LIN {X 0,Y 249.508,Z 932.66,A -85,B 0,C 180,E1 11833.837,E2 11833.837} C_VEL
LIN {X 0,Y 242.06,Z 946.637,A -85,B 0,C 180,E1 11830.431,E2 11830.431} C_VEL
LIN {X 0,Y 234.824,Z 959.705,A -85,B 0,C 180,E1 11826.415,E2 11826.415} C_VEL
LIN {X 0,Y 228.423,Z 971.273,A -85,B 0,C 180,E1 11821.878,E2 11821.878} C_VEL
LIN {X 0,Y 223.309,Z 980.961,A -85,B 0,C 180,E1 11817,E2 11817} C_VEL
LIN {X 0,Y 219.624,Z 988.763,A -85,B 0,C 180,E1 11811.922,E2 11811.922} C_VEL
LIN {X 0,Y 217.324,Z 994.963,A -85,B 0,C 180,E1 11806.575,E2 11806.575} C_VEL
LIN {X 0,Y 216.333,Z 999.398,A -85,B 0,C 180,E1 11801.195,E2 11801.195} C_VEL
LIN {X 0,Y 216.241,Z 1002.058,A -85,B 0,C 180,E1 11796.106,E2 11796.106} C_VEL
LIN {X 0,Y 216.392,Z 1003.045,A -85,B 0,C 180,E1 11791.59,E2 11791.59} C_VEL
LIN {X 0,Y 216.366,Z 1002.968,A -85,B 0,C 180,E1 11787.618,E2 11787.618} C_VEL
LIN {X 0,Y 216.189,Z 1001.566,A -85,B 0,C 180,E1 11782.828,E2 11782.828} C_VEL
LIN {X 0,Y 216.426,Z 998.664,A -85,B 0,C 180,E1 11777.732,E2 11777.732} C_VEL
LIN {X 0,Y 217.656,Z 993.876,A -85,B 0,C 180,E1 11772.352,E2 11772.352} C_VEL
LIN {X 0,Y 220.231,Z 987.265,A -85,B 0,C 180,E1 11767.019,E2 11767.019} C_VEL
LIN {X 0,Y 224.127,Z 979.16,A -85,B 0,C 180,E1 11762.042,E2 11762.042} C_VEL
LIN {X 0,Y 229.491,Z 969.097,A -85,B 0,C 180,E1 11757.231,E2 11757.231} C_VEL
LIN {X 0,Y 235.76,Z 957.78,A -85,B 0,C 180,E1 11752.972,E2 11752.972} C_VEL
LIN {X 0,Y 242.444,Z 945.727,A -85,B 0,C 180,E1 11749.339,E2 11749.339} C_VEL
LIN {X 0,Y 250.039,Z 931.432,A -85,B 0,C 180,E1 11745.911,E2 11745.911} C_VEL
LIN {X 0,Y 257.666,Z 916.125,A -85,B 0,C 180,E1 11742.993,E2 11742.993} C_VEL
LIN {X 0,Y 265.073,Z 899.972,A -85,B 0,C 180,E1 11740.532,E2 11740.532} C_VEL
LIN {X 0,Y 272.36,Z 882.29,A -85,B 0,C 180,E1 11738.394,E2 11738.394} C_VEL
LIN {X 0,Y 279.07,Z 863.665,A -85,B 0,C 180,E1 11736.627,E2 11736.627} C_VEL
LIN {X 0,Y 284.879,Z 844.815,A -85,B 0,C 180,E1 11735.245,E2 11735.245} C_VEL
LIN {X 0,Y 289.926,Z 824.777,A -85,B 0,C 180,E1 11734.141,E2 11734.141} C_VEL
LIN {X 0,Y 293.963,Z 803.375,A -85,B 0,C 180,E1 11733.295,E2 11733.295} C_VEL
LIN {X 0,Y 296.497,Z 782.175,A -85,B 0,C 180,E1 11732.711,E2 11732.711} C_VEL
LIN {X 0,Y 299.502,Z 753.951,A -85,B 0,C 180,E1 11732.36,E2 11732.36} C_VEL
LIN {X 0,Y 301.883,Z 735.107,A -85,B 0,C 180,E1 11732.253,E2 11732.253} C_VEL
LIN {X 0,Y 296.732,Z 710.347,A -85,B 0,C 180,E1 11729.497,E2 11729.497} C_VEL
LIN {X 0,Y 293.283,Z 686.164,A -85,B 0,C 180,E1 11727.059,E2 11727.059} C_VEL
LIN {X 0,Y 290.985,Z 658.881,A -85,B 0,C 180,E1 11724.649,E2 11724.649} C_VEL
LIN {X 0,Y 289.966,Z 631.512,A -85,B 0,C 180,E1 11722.557,E2 11722.557} C_VEL
LIN {X 0,Y 289.736,Z 625.924,A -85,B 0,C 180,E1 11722.095,E2 11722.095} C_VEL
LIN {X 0,Y 282.5,Z 605.873,A -85,B 0,C 180,E1 11716.553,E2 11716.553} C_VEL
LIN {X 0,Y 278.955,Z 593.643,A -85,B 0,C 180,E1 11712.629,E2 11712.629} C_VEL
LIN {X 0,Y 275.895,Z 578.468,A -85,B 0,C 180,E1 11706.817,E2 11706.817} C_VEL
LIN {X 0,Y 275.285,Z 568.562,A -85,B 0,C 180,E1 11702.289,E2 11702.289} C_VEL
LIN {X 0,Y 275.916,Z 561.635,A -85,B 0,C 180,E1 11698.65,E2 11698.65} C_VEL
LIN {X 0,Y 277.119,Z 556.907,A -85,B 0,C 180,E1 11695.758,E2 11695.758} C_VEL
LIN {X 0,Y 278.115,Z 554.651,A -85,B 0,C 180,E1 11694.015,E2 11694.015} C_VEL
LIN {X 0,Y 278.93,Z 555.456,A -85,B 0,C 180,E1 11692.378,E2 11692.378} C_VEL
LIN {X 0,Y 281.503,Z 559.555,A -85,B 0,C 180,E1 11688.527,E2 11688.527} C_VEL
LIN {X 0,Y 282.661,Z 561.038,A -85,B 0,C 180,E1 11687.227,E2 11687.227} C_VEL
LIN {X 0,Y 285.977,Z 565.926,A -85,B 0,C 180,E1 11684.07,E2 11684.07} C_VEL
LIN {X 0,Y 289.465,Z 571.159,A -85,B 0,C 180,E1 11681.366,E2 11681.366} C_VEL
LIN {X 0,Y 293.4,Z 577.167,A -85,B 0,C 180,E1 11678.772,E2 11678.772} C_VEL
LIN {X 0,Y 299.081,Z 586.337,A -85,B 0,C 180,E1 11675.562,E2 11675.562} C_VEL
LIN {X 0,Y 305.437,Z 597.593,A -85,B 0,C 180,E1 11672.458,E2 11672.458} C_VEL
LIN {X 0,Y 309.966,Z 606.51,A -85,B 0,C 180,E1 11670.461,E2 11670.461} C_VEL
LIN {X 0,Y 297.327,Z 772.309,A -85,B 0,C 180,E1 11666.864,E2 11666.864} C_VEL
LIN {X 0,Y 294.608,Z 792.529,A -85,B 0,C 180,E1 11666.172,E2 11666.172} C_VEL
LIN {X 0,Y 290.626,Z 813.159,A -85,B 0,C 180,E1 11665.173,E2 11665.173} C_VEL
LIN {X 0,Y 285.782,Z 832.475,A -85,B 0,C 180,E1 11663.918,E2 11663.918} C_VEL
LIN {X 0,Y 280.156,Z 850.837,A -85,B 0,C 180,E1 11662.389,E2 11662.389} C_VEL
LIN {X 0,Y 273.54,Z 869.084,A -85,B 0,C 180,E1 11660.465,E2 11660.465} C_VEL
LIN {X 0,Y 266.053,Z 886.914,A -85,B 0,C 180,E1 11658.081,E2 11658.081} C_VEL
LIN {X 0,Y 258.48,Z 902.921,A -85,B 0,C 180,E1 11655.376,E2 11655.376} C_VEL
LIN {X 0,Y 250.953,Z 917.393,A -85,B 0,C 180,E1 11652.324,E2 11652.324} C_VEL
LIN {X 0,Y 243.682,Z 930.447,A -85,B 0,C 180,E1 11648.885,E2 11648.885} C_VEL
LIN {X 0,Y 236.49,Z 942.746,A -85,B 0,C 180,E1 11644.802,E2 11644.802} C_VEL
LIN {X 0,Y 230.413,Z 952.929,A -85,B 0,C 180,E1 11640.51,E2 11640.51} C_VEL
LIN {X 0,Y 225.244,Z 961.693,A -85,B 0,C 180,E1 11635.785,E2 11635.785} C_VEL
LIN {X 0,Y 221.191,Z 968.962,A -85,B 0,C 180,E1 11630.644,E2 11630.644} C_VEL
LIN {X 0,Y 218.39,Z 974.6,A -85,B 0,C 180,E1 11625.126,E2 11625.126} C_VEL
LIN {X 0,Y 216.938,Z 978.219,A -85,B 0,C 180,E1 11619.817,E2 11619.817} C_VEL
LIN {X 0,Y 216.342,Z 980.279,A -85,B 0,C 180,E1 11614.505,E2 11614.505} C_VEL
LIN {X 0,Y 216.238,Z 980.863,A -85,B 0,C 180,E1 11609.469,E2 11609.469} C_VEL
LIN {X 0,Y 216.387,Z 980.118,A -85,B 0,C 180,E1 11604.696,E2 11604.696} C_VEL
LIN {X 0,Y 217.081,Z 977.836,A -85,B 0,C 180,E1 11599.382,E2 11599.382} C_VEL
LIN {X 0,Y 218.777,Z 973.736,A -85,B 0,C 180,E1 11593.811,E2 11593.811} C_VEL
LIN {X 0,Y 221.657,Z 968.101,A -85,B 0,C 180,E1 11588.568,E2 11588.568} C_VEL
LIN {X 0,Y 225.907,Z 960.633,A -85,B 0,C 180,E1 11583.446,E2 11583.446} C_VEL
LIN {X 0,Y 231.268,Z 951.656,A -85,B 0,C 180,E1 11578.746,E2 11578.746} C_VEL
LIN {X 0,Y 237.906,Z 940.55,A -85,B 0,C 180,E1 11574.253,E2 11574.253} C_VEL
LIN {X 0,Y 244.871,Z 928.525,A -85,B 0,C 180,E1 11570.431,E2 11570.431} C_VEL
LIN {X 0,Y 252.289,Z 915.077,A -85,B 0,C 180,E1 11567.025,E2 11567.025} C_VEL
LIN {X 0,Y 259.928,Z 900.139,A -85,B 0,C 180,E1 11563.999,E2 11563.999} C_VEL
LIN {X 0,Y 267.601,Z 883.56,A -85,B 0,C 180,E1 11561.32,E2 11561.32} C_VEL
LIN {X 0,Y 274.592,Z 866.606,A -85,B 0,C 180,E1 11559.14,E2 11559.14} C_VEL
LIN {X 0,Y 280.968,Z 848.815,A -85,B 0,C 180,E1 11557.31,E2 11557.31} C_VEL
LIN {X 0,Y 286.923,Z 828.967,A -85,B 0,C 180,E1 11555.711,E2 11555.711} C_VEL
LIN {X 0,Y 291.715,Z 808.912,A -85,B 0,C 180,E1 11554.478,E2 11554.478} C_VEL
LIN {X 0,Y 295.384,Z 788.518,A -85,B 0,C 180,E1 11553.556,E2 11553.556} C_VEL
LIN {X 0,Y 296.065,Z 783.376,A -85,B 0,C 180,E1 11553.352,E2 11553.352} C_VEL
LIN {X 0,Y 295.51,Z 784.886,A -85,B 0,C 180,E1 11553.294,E2 11553.294} C_VEL
LIN {X 0,Y 290.162,Z 799.608,A -85,B 0,C 180,E1 11552.949,E2 11552.949} C_VEL
LIN {X 0,Y 284.479,Z 812.877,A -85,B 0,C 180,E1 11552.694,E2 11552.694} C_VEL
LIN {X 0,Y 280.399,Z 820.06,A -85,B 0,C 180,E1 11552.37,E2 11552.37} C_VEL
LIN {X 0,Y 273.88,Z 829.294,A -85,B 0,C 180,E1 11551.593,E2 11551.593} C_VEL
LIN {X 0,Y 267.366,Z 836.64,A -85,B 0,C 180,E1 11550.571,E2 11550.571} C_VEL
LIN {X 0,Y 262.67,Z 841.252,A -85,B 0,C 180,E1 11549.66,E2 11549.66} C_VEL
LIN {X 0,Y 256.174,Z 848.136,A -85,B 0,C 180,E1 11548.573,E2 11548.573} C_VEL
LIN {X 0,Y 250.607,Z 852.992,A -85,B 0,C 180,E1 11547.311,E2 11547.311} C_VEL
LIN {X 0,Y 248.587,Z 854.447,A -85,B 0,C 180,E1 11546.775,E2 11546.775} C_VEL
LIN {X 0,Y 243.11,Z 859.517,A -85,B 0,C 180,E1 11545.585,E2 11545.585} C_VEL
LIN {X 0,Y 237.96,Z 863.392,A -85,B 0,C 180,E1 11544.053,E2 11544.053} C_VEL
LIN {X 0,Y 236.099,Z 864.688,A -85,B 0,C 180,E1 11543.459,E2 11543.459} C_VEL
LIN {X 0,Y 231.408,Z 868.479,A -85,B 0,C 180,E1 11542.081,E2 11542.081} C_VEL
LIN {X 0,Y 227.09,Z 871.222,A -85,B 0,C 180,E1 11540.308,E2 11540.308} C_VEL
LIN {X 0,Y 223.081,Z 874.46,A -85,B 0,C 180,E1 11538.827,E2 11538.827} C_VEL
LIN {X 0,Y 220.445,Z 875.936,A -85,B 0,C 180,E1 11537.419,E2 11537.419} C_VEL
LIN {X 0,Y 219.604,Z 876.415,A -85,B 0,C 180,E1 11536.942,E2 11536.942} C_VEL
LIN {X 0,Y 215.982,Z 879.302,A -85,B 0,C 180,E1 11535.3,E2 11535.3} C_VEL
LIN {X 0,Y 214.292,Z 880.186,A -85,B 0,C 180,E1 11534.042,E2 11534.042} C_VEL
LIN {X 0,Y 213.91,Z 880.409,A -85,B 0,C 180,E1 11533.516,E2 11533.516} C_VEL
LIN {X 0,Y 212.433,Z 891.843,A -85,B 0,C 180,E1 11529.756,E2 11529.756} C_VEL
LIN {X 0,Y 211.448,Z 902.388,A -85,B 0,C 180,E1 11525.427,E2 11525.427} C_VEL
LIN {X 0,Y 211.192,Z 910.701,A -85,B 0,C 180,E1 11521.086,E2 11521.086} C_VEL
LIN {X 0,Y 211.662,Z 917.257,A -85,B 0,C 180,E1 11516.751,E2 11516.751} C_VEL
LIN {X 0,Y 213.261,Z 922.908,A -85,B 0,C 180,E1 11511.604,E2 11511.604} C_VEL
LIN {X 0,Y 216.312,Z 926.54,A -85,B 0,C 180,E1 11506.365,E2 11506.365} C_VEL
LIN {X 0,Y 220.976,Z 928.025,A -85,B 0,C 180,E1 11501.261,E2 11501.261} C_VEL
LIN {X 0,Y 227.281,Z 927.461,A -85,B 0,C 180,E1 11496.402,E2 11496.402} C_VEL
LIN {X 0,Y 235.231,Z 924.927,A -85,B 0,C 180,E1 11491.849,E2 11491.849} C_VEL
LIN {X 0,Y 244.791,Z 920.464,A -85,B 0,C 180,E1 11487.651,E2 11487.651} C_VEL
LIN {X 0,Y 255.902,Z 914.126,A -85,B 0,C 180,E1 11483.844,E2 11483.844} C_VEL
LIN {X 0,Y 265.088,Z 908.328,A -85,B 0,C 180,E1 11481.246,E2 11481.246} C_VEL
LIN {X 0,Y 250.354,Z 921.045,A -85,B 0,C 180,E1 11477.635,E2 11477.635} C_VEL
LIN {X 0,Y 248.563,Z 923.055,A -85,B 0,C 180,E1 11477.065,E2 11477.065} C_VEL
LIN {X 0,Y 240.69,Z 937.7,A -85,B 0,C 180,E1 11473.929,E2 11473.929} C_VEL
LIN {X 0,Y 233.126,Z 950.904,A -85,B 0,C 180,E1 11470.365,E2 11470.365} C_VEL
LIN {X 0,Y 226.142,Z 962.79,A -85,B 0,C 180,E1 11466.334,E2 11466.334} C_VEL
LIN {X 0,Y 219.689,Z 973.857,A -85,B 0,C 180,E1 11461.562,E2 11461.562} C_VEL
LIN {X 0,Y 214.523,Z 983.296,A -85,B 0,C 180,E1 11456.283,E2 11456.283} C_VEL
LIN {X 0,Y 210.976,Z 990.727,A -85,B 0,C 180,E1 11450.822,E2 11450.822} C_VEL
LIN {X 0,Y 208.963,Z 996.327,A -85,B 0,C 180,E1 11445.26,E2 11445.26} C_VEL
LIN {X 0,Y 208.252,Z 999.989,A -85,B 0,C 180,E1 11439.955,E2 11439.955} C_VEL
LIN {X 0,Y 208.275,Z 1002.023,A -85,B 0,C 180,E1 11434.959,E2 11434.959} C_VEL
LIN {X 0,Y 208.42,Z 1002.729,A -85,B 0,C 180,E1 11430.551,E2 11430.551} C_VEL
LIN {X 0,Y 208.307,Z 1002.232,A -85,B 0,C 180,E1 11425.873,E2 11425.873} C_VEL
LIN {X 0,Y 208.203,Z 1000.547,A -85,B 0,C 180,E1 11421.162,E2 11421.162} C_VEL
LIN {X 0,Y 208.7,Z 997.166,A -85,B 0,C 180,E1 11415.859,E2 11415.859} C_VEL
LIN {X 0,Y 210.549,Z 991.635,A -85,B 0,C 180,E1 11410.008,E2 11410.008} C_VEL
LIN {X 0,Y 213.91,Z 984.361,A -85,B 0,C 180,E1 11404.437,E2 11404.437} C_VEL
LIN {X 0,Y 218.477,Z 975.891,A -85,B 0,C 180,E1 11399.472,E2 11399.472} C_VEL
LIN {X 0,Y 224.626,Z 965.286,A -85,B 0,C 180,E1 11394.645,E2 11394.645} C_VEL
LIN {X 0,Y 231.758,Z 953.089,A -85,B 0,C 180,E1 11390.321,E2 11390.321} C_VEL
LIN {X 0,Y 239.642,Z 939.321,A -85,B 0,C 180,E1 11386.496,E2 11386.496} C_VEL
LIN {X 0,Y 247.681,Z 924.434,A -85,B 0,C 180,E1 11383.228,E2 11383.228} C_VEL
LIN {X 0,Y 255.607,Z 908.668,A -85,B 0,C 180,E1 11380.492,E2 11380.492} C_VEL
LIN {X 0,Y 263.578,Z 891.117,A -85,B 0,C 180,E1 11378.084,E2 11378.084} C_VEL
LIN {X 0,Y 270.656,Z 873.481,A -85,B 0,C 180,E1 11376.18,E2 11376.18} C_VEL
LIN {X 0,Y 277.044,Z 855.14,A -85,B 0,C 180,E1 11374.63,E2 11374.63} C_VEL
LIN {X 0,Y 282.882,Z 835.046,A -85,B 0,C 180,E1 11373.34,E2 11373.34} C_VEL
LIN {X 0,Y 287.698,Z 813.932,A -85,B 0,C 180,E1 11372.359,E2 11372.359} C_VEL
LIN {X 0,Y 291.08,Z 792.615,A -85,B 0,C 180,E1 11371.65,E2 11371.65} C_VEL
LIN {X 0,Y 293.396,Z 770.364,A -85,B 0,C 180,E1 11371.208,E2 11371.208} C_VEL
LIN {X 0,Y 297.319,Z 737.114,A -85,B 0,C 180,E1 11370.937,E2 11370.937} C_VEL
LIN {X 0,Y 292.787,Z 713.367,A -85,B 0,C 180,E1 11368.269,E2 11368.269} C_VEL
LIN {X 0,Y 289.657,Z 689.519,A -85,B 0,C 180,E1 11365.822,E2 11365.822} C_VEL
LIN {X 0,Y 287.609,Z 661.966,A -85,B 0,C 180,E1 11363.348,E2 11363.348} C_VEL
LIN {X 0,Y 286.818,Z 634.141,A -85,B 0,C 180,E1 11361.189,E2 11361.189} C_VEL
LIN {X 0,Y 286.678,Z 630.805,A -85,B 0,C 180,E1 11360.892,E2 11360.892} C_VEL
LIN {X 0,Y 279.929,Z 610.615,A -85,B 0,C 180,E1 11355.167,E2 11355.167} C_VEL
LIN {X 0,Y 277.228,Z 600.398,A -85,B 0,C 180,E1 11351.81,E2 11351.81} C_VEL
LIN {X 0,Y 274.599,Z 585.5,A -85,B 0,C 180,E1 11346.061,E2 11346.061} C_VEL
LIN {X 0,Y 274.272,Z 575.732,A -85,B 0,C 180,E1 11341.566,E2 11341.566} C_VEL
LIN {X 0,Y 275.152,Z 568.696,A -85,B 0,C 180,E1 11337.836,E2 11337.836} C_VEL
LIN {X 0,Y 276.437,Z 564.313,A -85,B 0,C 180,E1 11335.124,E2 11335.124} C_VEL
LIN {X 0,Y 277.238,Z 562.671,A -85,B 0,C 180,E1 11333.788,E2 11333.788} C_VEL
LIN {X 0,Y 277.836,Z 563.406,A -85,B 0,C 180,E1 11332.556,E2 11332.556} C_VEL
LIN {X 0,Y 280.532,Z 567.621,A -85,B 0,C 180,E1 11328.487,E2 11328.487} C_VEL
LIN {X 0,Y 281.932,Z 569.872,A -85,B 0,C 180,E1 11326.881,E2 11326.881} C_VEL
LIN {X 0,Y 284.417,Z 573.484,A -85,B 0,C 180,E1 11324.503,E2 11324.503} C_VEL
LIN {X 0,Y 287.865,Z 578.85,A -85,B 0,C 180,E1 11321.731,E2 11321.731} C_VEL
LIN {X 0,Y 292.096,Z 585.427,A -85,B 0,C 180,E1 11318.883,E2 11318.883} C_VEL
LIN {X 0,Y 298.306,Z 596.028,A -85,B 0,C 180,E1 11315.336,E2 11315.336} C_VEL
LIN {X 0,Y 304.65,Z 607.99,A -85,B 0,C 180,E1 11312.222,E2 11312.222} C_VEL
LIN {X 0,Y 305.805,Z 610.542,A -85,B 0,C 180,E1 11311.685,E2 11311.685} C_VEL
LIN {X 0,Y 293.023,Z 772.739,A -85,B 0,C 180,E1 11308.171,E2 11308.171} C_VEL
LIN {X 0,Y 290.201,Z 793.084,A -85,B 0,C 180,E1 11307.476,E2 11307.476} C_VEL
LIN {X 0,Y 286.122,Z 813.58,A -85,B 0,C 180,E1 11306.486,E2 11306.486} C_VEL
LIN {X 0,Y 281.137,Z 832.867,A -85,B 0,C 180,E1 11305.238,E2 11305.238} C_VEL
LIN {X 0,Y 275.272,Z 851.399,A -85,B 0,C 180,E1 11303.696,E2 11303.696} C_VEL
LIN {X 0,Y 268.495,Z 869.487,A -85,B 0,C 180,E1 11301.788,E2 11301.788} C_VEL
LIN {X 0,Y 260.738,Z 887.322,A -85,B 0,C 180,E1 11299.399,E2 11299.399} C_VEL
LIN {X 0,Y 252.873,Z 903.332,A -85,B 0,C 180,E1 11296.678,E2 11296.678} C_VEL
LIN {X 0,Y 245.032,Z 917.806,A -85,B 0,C 180,E1 11293.597,E2 11293.597} C_VEL
LIN {X 0,Y 237.425,Z 930.862,A -85,B 0,C 180,E1 11290.113,E2 11290.113} C_VEL
LIN {X 0,Y 229.872,Z 943.163,A -85,B 0,C 180,E1 11285.957,E2 11285.957} C_VEL
LIN {X 0,Y 223.453,Z 953.346,A -85,B 0,C 180,E1 11281.567,E2 11281.567} C_VEL
LIN {X 0,Y 217.962,Z 962.111,A -85,B 0,C 180,E1 11276.714,E2 11276.714} C_VEL
LIN {X 0,Y 213.539,Z 969.52,A -85,B 0,C 180,E1 11271.285,E2 11271.285} C_VEL
LIN {X 0,Y 210.601,Z 975.016,A -85,B 0,C 180,E1 11265.699,E2 11265.699} C_VEL
LIN {X 0,Y 209.02,Z 978.633,A -85,B 0,C 180,E1 11260.193,E2 11260.193} C_VEL
LIN {X 0,Y 208.363,Z 980.691,A -85,B 0,C 180,E1 11254.678,E2 11254.678} C_VEL
LIN {X 0,Y 208.249,Z 981.275,A -85,B 0,C 180,E1 11249.448,E2 11249.448} C_VEL
LIN {X 0,Y 208.411,Z 980.53,A -85,B 0,C 180,E1 11244.492,E2 11244.492} C_VEL
LIN {X 0,Y 209.173,Z 978.25,A -85,B 0,C 180,E1 11238.976,E2 11238.976} C_VEL
LIN {X 0,Y 211.021,Z 974.151,A -85,B 0,C 180,E1 11233.199,E2 11233.199} C_VEL
LIN {X 0,Y 214.126,Z 968.516,A -85,B 0,C 180,E1 11227.774,E2 11227.774} C_VEL
LIN {X 0,Y 218.67,Z 961.049,A -85,B 0,C 180,E1 11222.494,E2 11222.494} C_VEL
LIN {X 0,Y 224.361,Z 952.07,A -85,B 0,C 180,E1 11217.67,E2 11217.67} C_VEL
LIN {X 0,Y 231.368,Z 940.962,A -85,B 0,C 180,E1 11213.079,E2 11213.079} C_VEL
LIN {X 0,Y 238.677,Z 928.935,A -85,B 0,C 180,E1 11209.191,E2 11209.191} C_VEL
LIN {X 0,Y 246.432,Z 915.484,A -85,B 0,C 180,E1 11205.742,E2 11205.742} C_VEL
LIN {X 0,Y 254.384,Z 900.542,A -85,B 0,C 180,E1 11202.691,E2 11202.691} C_VEL
LIN {X 0,Y 262.351,Z 883.958,A -85,B 0,C 180,E1 11199.999,E2 11199.999} C_VEL
LIN {X 0,Y 269.59,Z 866.998,A -85,B 0,C 180,E1 11197.815,E2 11197.815} C_VEL
LIN {X 0,Y 276.178,Z 849.2,A -85,B 0,C 180,E1 11195.986,E2 11195.986} C_VEL
LIN {X 0,Y 281.983,Z 830.511,A -85,B 0,C 180,E1 11194.475,E2 11194.475} C_VEL
LIN {X 0,Y 286.783,Z 811.098,A -85,B 0,C 180,E1 11193.247,E2 11193.247} C_VEL
LIN {X 0,Y 281.294,Z 818.614,A -85,B 0,C 180,E1 11192.462,E2 11192.462} C_VEL
LIN {X 0,Y 280.399,Z 820.06,A -85,B 0,C 180,E1 11192.37,E2 11192.37} C_VEL
LIN {X 0,Y 277.511,Z 825.438,A -85,B 0,C 180,E1 11192.229,E2 11192.229} C_VEL
LIN {X 0,Y 272.262,Z 836.502,A -85,B 0,C 180,E1 11192.306,E2 11192.306} C_VEL
LIN {X 0,Y 269.365,Z 840.573,A -85,B 0,C 180,E1 11192.061,E2 11192.061} C_VEL
LIN {X 0,Y 268.908,Z 841.051,A -85,B 0,C 180,E1 11191.993,E2 11191.993} C_VEL
LIN {X 0,Y 262.599,Z 846.992,A -85,B 0,C 180,E1 11190.932,E2 11190.932} C_VEL
LIN {X 0,Y 255.547,Z 854.023,A -85,B 0,C 180,E1 11189.796,E2 11189.796} C_VEL
LIN {X 0,Y 248.708,Z 859.476,A -85,B 0,C 180,E1 11188.32,E2 11188.32} C_VEL
LIN {X 0,Y 240.057,Z 866.645,A -85,B 0,C 180,E1 11186.425,E2 11186.425} C_VEL
LIN {X 0,Y 234.278,Z 870.564,A -85,B 0,C 180,E1 11184.724,E2 11184.724} C_VEL
LIN {X 0,Y 228.811,Z 874.703,A -85,B 0,C 180,E1 11183.159,E2 11183.159} C_VEL
LIN {X 0,Y 224.301,Z 877.414,A -85,B 0,C 180,E1 11181.441,E2 11181.441} C_VEL
LIN {X 0,Y 219.526,Z 880.861,A -85,B 0,C 180,E1 11179.697,E2 11179.697} C_VEL
LIN {X 0,Y 216.358,Z 882.596,A -85,B 0,C 180,E1 11178.037,E2 11178.037} C_VEL
LIN {X 0,Y 212.19,Z 885.615,A -85,B 0,C 180,E1 11176.142,E2 11176.142} C_VEL
LIN {X 0,Y 209.664,Z 886.901,A -85,B 0,C 180,E1 11174.359,E2 11174.359} C_VEL
LIN {X 0,Y 206.503,Z 889.328,A -85,B 0,C 180,E1 11172.585,E2 11172.585} C_VEL
LIN {X 0,Y 204.863,Z 890.186,A -85,B 0,C 180,E1 11170.973,E2 11170.973} C_VEL
LIN {X 0,Y 204.663,Z 890.482,A -85,B 0,C 180,E1 11170.55,E2 11170.55} C_VEL
LIN {X 0,Y 203.56,Z 901.222,A -85,B 0,C 180,E1 11166.204,E2 11166.204} C_VEL
LIN {X 0,Y 203.2,Z 910.642,A -85,B 0,C 180,E1 11161.41,E2 11161.41} C_VEL
LIN {X 0,Y 203.695,Z 917.877,A -85,B 0,C 180,E1 11156.624,E2 11156.624} C_VEL
LIN {X 0,Y 205.138,Z 923.3,A -85,B 0,C 180,E1 11151.875,E2 11151.875} C_VEL
LIN {X 0,Y 208.043,Z 927.408,A -85,B 0,C 180,E1 11146.663,E2 11146.663} C_VEL
LIN {X 0,Y 212.457,Z 929.549,A -85,B 0,C 180,E1 11141.621,E2 11141.621} C_VEL
LIN {X 0,Y 219.133,Z 929.77,A -85,B 0,C 180,E1 11136.327,E2 11136.327} C_VEL
LIN {X 0,Y 227.244,Z 928.012,A -85,B 0,C 180,E1 11131.629,E2 11131.629} C_VEL
LIN {X 0,Y 237.008,Z 924.384,A -85,B 0,C 180,E1 11127.318,E2 11127.318} C_VEL
LIN {X 0,Y 248.351,Z 918.964,A -85,B 0,C 180,E1 11123.428,E2 11123.428} C_VEL
LIN {X 0,Y 255.207,Z 915.31,A -85,B 0,C 180,E1 11121.428,E2 11121.428} C_VEL
LIN {X 0,Y 240.796,Z 926.761,A -85,B 0,C 180,E1 11117.658,E2 11117.658} C_VEL
LIN {X 0,Y 232.275,Z 941.595,A -85,B 0,C 180,E1 11114.217,E2 11114.217} C_VEL
LIN {X 0,Y 224.185,Z 954.904,A -85,B 0,C 180,E1 11110.295,E2 11110.295} C_VEL
LIN {X 0,Y 217.245,Z 966.132,A -85,B 0,C 180,E1 11106.096,E2 11106.096} C_VEL
LIN {X 0,Y 211.155,Z 976.06,A -85,B 0,C 180,E1 11101.392,E2 11101.392} C_VEL
LIN {X 0,Y 206.035,Z 984.955,A -85,B 0,C 180,E1 11095.899,E2 11095.899} C_VEL
LIN {X 0,Y 202.623,Z 991.877,A -85,B 0,C 180,E1 11090.209,E2 11090.209} C_VEL
LIN {X 0,Y 200.773,Z 996.99,A -85,B 0,C 180,E1 11084.42,E2 11084.42} C_VEL
LIN {X 0,Y 200.225,Z 1000.394,A -85,B 0,C 180,E1 11078.606,E2 11078.606} C_VEL
LIN {X 0,Y 200.334,Z 1001.972,A -85,B 0,C 180,E1 11073.722,E2 11073.722} C_VEL
LIN {X 0,Y 200.426,Z 1002.291,A -85,B 0,C 180,E1 11069.144,E2 11069.144} C_VEL
LIN {X 0,Y 200.262,Z 1001.527,A -85,B 0,C 180,E1 11064.558,E2 11064.558} C_VEL
LIN {X 0,Y 200.299,Z 999.213,A -85,B 0,C 180,E1 11059.067,E2 11059.067} C_VEL
LIN {X 0,Y 201.3,Z 995.149,A -85,B 0,C 180,E1 11053.258,E2 11053.258} C_VEL
LIN {X 0,Y 203.742,Z 989.322,A -85,B 0,C 180,E1 11047.495,E2 11047.495} C_VEL
LIN {X 0,Y 207.843,Z 981.57,A -85,B 0,C 180,E1 11041.874,E2 11041.874} C_VEL
LIN {X 0,Y 213.318,Z 972.31,A -85,B 0,C 180,E1 11036.744,E2 11036.744} C_VEL
LIN {X 0,Y 219.907,Z 961.632,A -85,B 0,C 180,E1 11032.136,E2 11032.136} C_VEL
LIN {X 0,Y 227.808,Z 948.812,A -85,B 0,C 180,E1 11027.817,E2 11027.817} C_VEL
LIN {X 0,Y 235.84,Z 935.273,A -85,B 0,C 180,E1 11024.237,E2 11024.237} C_VEL
LIN {X 0,Y 243.881,Z 920.882,A -85,B 0,C 180,E1 11021.211,E2 11021.211} C_VEL
LIN {X 0,Y 252.416,Z 904.235,A -85,B 0,C 180,E1 11018.455,E2 11018.455} C_VEL
LIN {X 0,Y 260.607,Z 886.289,A -85,B 0,C 180,E1 11016.138,E2 11016.138} C_VEL
LIN {X 0,Y 267.867,Z 868.033,A -85,B 0,C 180,E1 11014.307,E2 11014.307} C_VEL
LIN {X 0,Y 274.307,Z 849.121,A -85,B 0,C 180,E1 11012.843,E2 11012.843} C_VEL
LIN {X 0,Y 279.734,Z 829.887,A -85,B 0,C 180,E1 11011.715,E2 11011.715} C_VEL
LIN {X 0,Y 284.262,Z 809.32,A -85,B 0,C 180,E1 11010.833,E2 11010.833} C_VEL
LIN {X 0,Y 287.374,Z 788.684,A -85,B 0,C 180,E1 11010.188,E2 11010.188} C_VEL
LIN {X 0,Y 290.015,Z 763.795,A -85,B 0,C 180,E1 11009.782,E2 11009.782} C_VEL
LIN {X 0,Y 292.967,Z 739.242,A -85,B 0,C 180,E1 11009.604,E2 11009.604} C_VEL
LIN {X 0,Y 288.979,Z 716.38,A -85,B 0,C 180,E1 11007.008,E2 11007.008} C_VEL
LIN {X 0,Y 286.193,Z 693.135,A -85,B 0,C 180,E1 11004.58,E2 11004.58} C_VEL
LIN {X 0,Y 284.392,Z 665.207,A -85,B 0,C 180,E1 11002.029,E2 11002.029} C_VEL
LIN {X 0,Y 283.838,Z 636.802,A -85,B 0,C 180,E1 10999.795,E2 10999.795} C_VEL
LIN {X 0,Y 283.748,Z 635.704,A -85,B 0,C 180,E1 10999.665,E2 10999.665} C_VEL
LIN {X 0,Y 277.479,Z 615.226,A -85,B 0,C 180,E1 10993.705,E2 10993.705} C_VEL
LIN {X 0,Y 275.525,Z 607.017,A -85,B 0,C 180,E1 10990.93,E2 10990.93} C_VEL
LIN {X 0,Y 273.352,Z 592.532,A -85,B 0,C 180,E1 10985.299,E2 10985.299} C_VEL
LIN {X 0,Y 273.304,Z 582.898,A -85,B 0,C 180,E1 10980.838,E2 10980.838} C_VEL
LIN {X 0,Y 274.375,Z 576.023,A -85,B 0,C 180,E1 10977.18,E2 10977.18} C_VEL
LIN {X 0,Y 275.791,Z 571.713,A -85,B 0,C 180,E1 10974.487,E2 10974.487} C_VEL
LIN {X 0,Y 276.364,Z 570.698,A -85,B 0,C 180,E1 10973.56,E2 10973.56} C_VEL
LIN {X 0,Y 276.985,Z 571.976,A -85,B 0,C 180,E1 10972.22,E2 10972.22} C_VEL
LIN {X 0,Y 279.968,Z 576.461,A -85,B 0,C 180,E1 10967.94,E2 10967.94} C_VEL
LIN {X 0,Y 282.978,Z 581.232,A -85,B 0,C 180,E1 10964.843,E2 10964.843} C_VEL
LIN {X 0,Y 286.153,Z 586.321,A -85,B 0,C 180,E1 10962.197,E2 10962.197} C_VEL
LIN {X 0,Y 290.187,Z 592.853,A -85,B 0,C 180,E1 10959.371,E2 10959.371} C_VEL
LIN {X 0,Y 295.901,Z 602.927,A -85,B 0,C 180,E1 10955.972,E2 10955.972} C_VEL
LIN {X 0,Y 301.789,Z 614.395,A -85,B 0,C 180,E1 10952.95,E2 10952.95} C_VEL
LIN {X 0,Y 288.876,Z 773.17,A -85,B 0,C 180,E1 10949.516,E2 10949.516} C_VEL
LIN {X 0,Y 285.98,Z 793.448,A -85,B 0,C 180,E1 10948.828,E2 10948.828} C_VEL
LIN {X 0,Y 281.772,Z 814.005,A -85,B 0,C 180,E1 10947.841,E2 10947.841} C_VEL
LIN {X 0,Y 276.647,Z 833.259,A -85,B 0,C 180,E1 10946.602,E2 10946.602} C_VEL
LIN {X 0,Y 270.54,Z 851.956,A -85,B 0,C 180,E1 10945.051,E2 10945.051} C_VEL
LIN {X 0,Y 263.598,Z 869.891,A -85,B 0,C 180,E1 10943.161,E2 10943.161} C_VEL
LIN {X 0,Y 255.565,Z 887.73,A -85,B 0,C 180,E1 10940.771,E2 10940.771} C_VEL
LIN {X 0,Y 247.402,Z 903.743,A -85,B 0,C 180,E1 10938.039,E2 10938.039} C_VEL
LIN {X 0,Y 239.239,Z 918.219,A -85,B 0,C 180,E1 10934.933,E2 10934.933} C_VEL
LIN {X 0,Y 231.282,Z 931.277,A -85,B 0,C 180,E1 10931.408,E2 10931.408} C_VEL
LIN {X 0,Y 223.319,Z 943.632,A -85,B 0,C 180,E1 10927.159,E2 10927.159} C_VEL
LIN {X 0,Y 216.573,Z 953.764,A -85,B 0,C 180,E1 10922.693,E2 10922.693} C_VEL
LIN {X 0,Y 210.741,Z 962.529,A -85,B 0,C 180,E1 10917.706,E2 10917.706} C_VEL
LIN {X 0,Y 206.096,Z 969.797,A -85,B 0,C 180,E1 10912.234,E2 10912.234} C_VEL
LIN {X 0,Y 202.831,Z 975.433,A -85,B 0,C 180,E1 10906.317,E2 10906.317} C_VEL
LIN {X 0,Y 201.107,Z 979.048,A -85,B 0,C 180,E1 10900.599,E2 10900.599} C_VEL
LIN {X 0,Y 200.385,Z 981.104,A -85,B 0,C 180,E1 10894.864,E2 10894.864} C_VEL
LIN {X 0,Y 200.261,Z 981.708,A -85,B 0,C 180,E1 10889.712,E2 10889.712} C_VEL
LIN {X 0,Y 200.418,Z 981.006,A -85,B 0,C 180,E1 10884.559,E2 10884.559} C_VEL
LIN {X 0,Y 201.212,Z 978.815,A -85,B 0,C 180,E1 10878.824,E2 10878.824} C_VEL
LIN {X 0,Y 203.037,Z 975.054,A -85,B 0,C 180,E1 10873.108,E2 10873.108} C_VEL
LIN {X 0,Y 206.241,Z 969.613,A -85,B 0,C 180,E1 10867.479,E2 10867.479} C_VEL
LIN {X 0,Y 210.944,Z 962.31,A -85,B 0,C 180,E1 10862.013,E2 10862.013} C_VEL
LIN {X 0,Y 216.835,Z 953.484,A -85,B 0,C 180,E1 10857.034,E2 10857.034} C_VEL
LIN {X 0,Y 223.67,Z 943.23,A -85,B 0,C 180,E1 10852.557,E2 10852.557} C_VEL
LIN {X 0,Y 231.175,Z 931.599,A -85,B 0,C 180,E1 10848.565,E2 10848.565} C_VEL
LIN {X 0,Y 239.124,Z 918.605,A -85,B 0,C 180,E1 10845.036,E2 10845.036} C_VEL
LIN {X 0,Y 247.283,Z 904.203,A -85,B 0,C 180,E1 10841.927,E2 10841.927} C_VEL
LIN {X 0,Y 255.442,Z 888.255,A -85,B 0,C 180,E1 10839.192,E2 10839.192} C_VEL
LIN {X 0,Y 263.082,Z 871.37,A -85,B 0,C 180,E1 10836.905,E2 10836.905} C_VEL
LIN {X 0,Y 269.89,Z 854.075,A -85,B 0,C 180,E1 10835.04,E2 10835.04} C_VEL
LIN {X 0,Y 276.185,Z 835.276,A -85,B 0,C 180,E1 10833.438,E2 10833.438} C_VEL
LIN {X 0,Y 277.289,Z 831.551,A -85,B 0,C 180,E1 10833.149,E2 10833.149} C_VEL
LIN {X 0,Y 270.204,Z 839.72,A -85,B 0,C 180,E1 10832.199,E2 10832.199} C_VEL
LIN {X 0,Y 268.908,Z 841.051,A -85,B 0,C 180,E1 10831.993,E2 10831.993} C_VEL
LIN {X 0,Y 265.735,Z 844.925,A -85,B 0,C 180,E1 10831.639,E2 10831.639} C_VEL
LIN {X 0,Y 257.625,Z 856.885,A -85,B 0,C 180,E1 10831.367,E2 10831.367} C_VEL
LIN {X 0,Y 254.758,Z 859.916,A -85,B 0,C 180,E1 10831.017,E2 10831.017} C_VEL
LIN {X 0,Y 247.46,Z 865.376,A -85,B 0,C 180,E1 10829.534,E2 10829.534} C_VEL
LIN {X 0,Y 239.384,Z 871.846,A -85,B 0,C 180,E1 10827.892,E2 10827.892} C_VEL
LIN {X 0,Y 231.661,Z 876.9,A -85,B 0,C 180,E1 10825.844,E2 10825.844} C_VEL
LIN {X 0,Y 225.478,Z 881.169,A -85,B 0,C 180,E1 10824.077,E2 10824.077} C_VEL
LIN {X 0,Y 221.368,Z 883.564,A -85,B 0,C 180,E1 10822.577,E2 10822.577} C_VEL
LIN {X 0,Y 215.873,Z 887.114,A -85,B 0,C 180,E1 10820.611,E2 10820.611} C_VEL
LIN {X 0,Y 212.411,Z 888.997,A -85,B 0,C 180,E1 10818.954,E2 10818.954} C_VEL
LIN {X 0,Y 207.877,Z 891.97,A -85,B 0,C 180,E1 10816.826,E2 10816.826} C_VEL
LIN {X 0,Y 205.481,Z 893.224,A -85,B 0,C 180,E1 10815.234,E2 10815.234} C_VEL
LIN {X 0,Y 201.917,Z 895.647,A -85,B 0,C 180,E1 10813.167,E2 10813.167} C_VEL
LIN {X 0,Y 199.812,Z 896.772,A -85,B 0,C 180,E1 10811.242,E2 10811.242} C_VEL
LIN {X 0,Y 196.93,Z 898.995,A -85,B 0,C 180,E1 10809.056,E2 10809.056} C_VEL
LIN {X 0,Y 195.702,Z 899.845,A -85,B 0,C 180,E1 10807.044,E2 10807.044} C_VEL
LIN {X 0,Y 195.207,Z 909.347,A -85,B 0,C 180,E1 10802.349,E2 10802.349} C_VEL
LIN {X 0,Y 195.617,Z 917.672,A -85,B 0,C 180,E1 10797.071,E2 10797.071} C_VEL
LIN {X 0,Y 197.136,Z 923.871,A -85,B 0,C 180,E1 10791.836,E2 10791.836} C_VEL
LIN {X 0,Y 199.939,Z 928.226,A -85,B 0,C 180,E1 10786.701,E2 10786.701} C_VEL
LIN {X 0,Y 204.45,Z 930.955,A -85,B 0,C 180,E1 10781.466,E2 10781.466} C_VEL
LIN {X 0,Y 210.941,Z 931.844,A -85,B 0,C 180,E1 10776.241,E2 10776.241} C_VEL
LIN {X 0,Y 219.203,Z 930.841,A -85,B 0,C 180,E1 10771.384,E2 10771.384} C_VEL
LIN {X 0,Y 229.708,Z 927.828,A -85,B 0,C 180,E1 10766.74,E2 10766.74} C_VEL
LIN {X 0,Y 241.359,Z 923.207,A -85,B 0,C 180,E1 10762.784,E2 10762.784} C_VEL
LIN {X 0,Y 245.211,Z 921.502,A -85,B 0,C 180,E1 10761.613,E2 10761.613} C_VEL
LIN {X 0,Y 233.058,Z 930.342,A -85,B 0,C 180,E1 10758.289,E2 10758.289} C_VEL
LIN {X 0,Y 224.376,Z 944.595,A -85,B 0,C 180,E1 10754.757,E2 10754.757} C_VEL
LIN {X 0,Y 215.905,Z 957.711,A -85,B 0,C 180,E1 10750.582,E2 10750.582} C_VEL
LIN {X 0,Y 208.704,Z 968.635,A -85,B 0,C 180,E1 10746.107,E2 10746.107} C_VEL
LIN {X 0,Y 202.324,Z 978.468,A -85,B 0,C 180,E1 10740.929,E2 10740.929} C_VEL
LIN {X 0,Y 197.34,Z 986.769,A -85,B 0,C 180,E1 10735.19,E2 10735.19} C_VEL
LIN {X 0,Y 194.147,Z 993.172,A -85,B 0,C 180,E1 10729.246,E2 10729.246} C_VEL
LIN {X 0,Y 192.558,Z 997.807,A -85,B 0,C 180,E1 10723.209,E2 10723.209} C_VEL
LIN {X 0,Y 192.224,Z 1000.577,A -85,B 0,C 180,E1 10717.473,E2 10717.473} C_VEL
LIN {X 0,Y 192.393,Z 1001.76,A -85,B 0,C 180,E1 10712.384,E2 10712.384} C_VEL
LIN {X 0,Y 192.414,Z 1001.807,A -85,B 0,C 180,E1 10708.215,E2 10708.215} C_VEL
LIN {X 0,Y 192.212,Z 1000.799,A -85,B 0,C 180,E1 10703.13,E2 10703.13} C_VEL
LIN {X 0,Y 192.456,Z 998.121,A -85,B 0,C 180,E1 10697.398,E2 10697.398} C_VEL
LIN {X 0,Y 193.892,Z 993.669,A -85,B 0,C 180,E1 10691.356,E2 10691.356} C_VEL
LIN {X 0,Y 197.11,Z 987.088,A -85,B 0,C 180,E1 10685.102,E2 10685.102} C_VEL
LIN {X 0,Y 201.99,Z 978.872,A -85,B 0,C 180,E1 10679.348,E2 10679.348} C_VEL
LIN {X 0,Y 208.064,Z 969.469,A -85,B 0,C 180,E1 10674.304,E2 10674.304} C_VEL
LIN {X 0,Y 215.204,Z 958.623,A -85,B 0,C 180,E1 10669.776,E2 10669.776} C_VEL
LIN {X 0,Y 223.291,Z 946.049,A -85,B 0,C 180,E1 10665.692,E2 10665.692} C_VEL
LIN {X 0,Y 231.87,Z 932.049,A -85,B 0,C 180,E1 10662.126,E2 10662.126} C_VEL
LIN {X 0,Y 240.392,Z 917.115,A -85,B 0,C 180,E1 10659.133,E2 10659.133} C_VEL
LIN {X 0,Y 248.912,Z 900.749,A -85,B 0,C 180,E1 10656.548,E2 10656.548} C_VEL
LIN {X 0,Y 256.925,Z 883.509,A -85,B 0,C 180,E1 10654.411,E2 10654.411} C_VEL
LIN {X 0,Y 264.248,Z 865.462,A -85,B 0,C 180,E1 10652.661,E2 10652.661} C_VEL
LIN {X 0,Y 270.759,Z 846.477,A -85,B 0,C 180,E1 10651.255,E2 10651.255} C_VEL
LIN {X 0,Y 276.157,Z 827.306,A -85,B 0,C 180,E1 10650.186,E2 10650.186} C_VEL
LIN {X 0,Y 280.65,Z 806.664,A -85,B 0,C 180,E1 10649.343,E2 10649.343} C_VEL
LIN {X 0,Y 283.807,Z 784.843,A -85,B 0,C 180,E1 10648.705,E2 10648.705} C_VEL
LIN {X 0,Y 286.934,Z 756.65,A -85,B 0,C 180,E1 10648.338,E2 10648.338} C_VEL
LIN {X 0,Y 288.781,Z 741.288,A -85,B 0,C 180,E1 10648.229,E2 10648.229} C_VEL
LIN {X 0,Y 285.037,Z 717.476,A -85,B 0,C 180,E1 10645.49,E2 10645.49} C_VEL
LIN {X 0,Y 282.535,Z 692.007,A -85,B 0,C 180,E1 10642.854,E2 10642.854} C_VEL
LIN {X 0,Y 281.274,Z 666.026,A -85,B 0,C 180,E1 10640.482,E2 10640.482} C_VEL
LIN {X 0,Y 280.944,Z 640.642,A -85,B 0,C 180,E1 10638.412,E2 10638.412} C_VEL
LIN {X 0,Y 275.317,Z 620.329,A -85,B 0,C 180,E1 10632.372,E2 10632.372} C_VEL
LIN {X 0,Y 273.805,Z 613.228,A -85,B 0,C 180,E1 10629.882,E2 10629.882} C_VEL
LIN {X 0,Y 272.155,Z 599.562,A -85,B 0,C 180,E1 10624.53,E2 10624.53} C_VEL
LIN {X 0,Y 272.38,Z 590.061,A -85,B 0,C 180,E1 10620.105,E2 10620.105} C_VEL
LIN {X 0,Y 273.726,Z 583.021,A -85,B 0,C 180,E1 10616.335,E2 10616.335} C_VEL
LIN {X 0,Y 275.393,Z 578.658,A -85,B 0,C 180,E1 10613.537,E2 10613.537} C_VEL
LIN {X 0,Y 278.639,Z 584.168,A -85,B 0,C 180,E1 10608.302,E2 10608.302} C_VEL
LIN {X 0,Y 281.551,Z 588.975,A -85,B 0,C 180,E1 10605.185,E2 10605.185} C_VEL
LIN {X 0,Y 284.459,Z 593.791,A -85,B 0,C 180,E1 10602.669,E2 10602.669} C_VEL
LIN {X 0,Y 288.3,Z 600.273,A -85,B 0,C 180,E1 10599.866,E2 10599.866} C_VEL
LIN {X 0,Y 293.533,Z 609.824,A -85,B 0,C 180,E1 10596.619,E2 10596.619} C_VEL
LIN {X 0,Y 297.909,Z 618.724,A -85,B 0,C 180,E1 10594.229,E2 10594.229} C_VEL
LIN {X 0,Y 284.882,Z 773.699,A -85,B 0,C 180,E1 10590.896,E2 10590.896} C_VEL
LIN {X 0,Y 281.892,Z 793.997,A -85,B 0,C 180,E1 10590.211,E2 10590.211} C_VEL
LIN {X 0,Y 277.585,Z 814.428,A -85,B 0,C 180,E1 10589.237,E2 10589.237} C_VEL
LIN {X 0,Y 272.318,Z 833.653,A -85,B 0,C 180,E1 10588.009,E2 10588.009} C_VEL
LIN {X 0,Y 266.17,Z 851.979,A -85,B 0,C 180,E1 10586.503,E2 10586.503} C_VEL
LIN {X 0,Y 258.859,Z 870.295,A -85,B 0,C 180,E1 10584.585,E2 10584.585} C_VEL
LIN {X 0,Y 250.725,Z 887.762,A -85,B 0,C 180,E1 10582.253,E2 10582.253} C_VEL
LIN {X 0,Y 242.37,Z 903.611,A -85,B 0,C 180,E1 10579.562,E2 10579.562} C_VEL
LIN {X 0,Y 234.129,Z 917.727,A -85,B 0,C 180,E1 10576.55,E2 10576.55} C_VEL
LIN {X 0,Y 225.76,Z 930.942,A -85,B 0,C 180,E1 10573.002,E2 10573.002} C_VEL
LIN {X 0,Y 217.817,Z 942.76,A -85,B 0,C 180,E1 10568.966,E2 10568.966} C_VEL
LIN {X 0,Y 210.522,Z 953.184,A -85,B 0,C 180,E1 10564.413,E2 10564.413} C_VEL
LIN {X 0,Y 203.877,Z 962.556,A -85,B 0,C 180,E1 10559.045,E2 10559.045} C_VEL
LIN {X 0,Y 198.613,Z 970.215,A -85,B 0,C 180,E1 10553.119,E2 10553.119} C_VEL
LIN {X 0,Y 195.085,Z 975.85,A -85,B 0,C 180,E1 10546.984,E2 10546.984} C_VEL
LIN {X 0,Y 193.206,Z 979.463,A -85,B 0,C 180,E1 10541.037,E2 10541.037} C_VEL
LIN {X 0,Y 192.409,Z 981.516,A -85,B 0,C 180,E1 10535.067,E2 10535.067} C_VEL
LIN {X 0,Y 192.272,Z 982.12,A -85,B 0,C 180,E1 10529.7,E2 10529.7} C_VEL
LIN {X 0,Y 192.444,Z 981.418,A -85,B 0,C 180,E1 10524.333,E2 10524.333} C_VEL
LIN {X 0,Y 193.315,Z 979.229,A -85,B 0,C 180,E1 10518.361,E2 10518.361} C_VEL
LIN {X 0,Y 195.311,Z 975.47,A -85,B 0,C 180,E1 10512.418,E2 10512.418} C_VEL
LIN {X 0,Y 198.771,Z 970.029,A -85,B 0,C 180,E1 10506.583,E2 10506.583} C_VEL
LIN {X 0,Y 204.037,Z 962.411,A -85,B 0,C 180,E1 10500.724,E2 10500.724} C_VEL
LIN {X 0,Y 210.809,Z 952.899,A -85,B 0,C 180,E1 10495.307,E2 10495.307} C_VEL
LIN {X 0,Y 218.605,Z 941.787,A -85,B 0,C 180,E1 10490.522,E2 10490.522} C_VEL
LIN {X 0,Y 226.656,Z 929.755,A -85,B 0,C 180,E1 10486.513,E2 10486.513} C_VEL
LIN {X 0,Y 235.114,Z 916.298,A -85,B 0,C 180,E1 10482.99,E2 10482.99} C_VEL
LIN {X 0,Y 243.724,Z 901.349,A -85,B 0,C 180,E1 10479.899,E2 10479.899} C_VEL
LIN {X 0,Y 252.298,Z 884.755,A -85,B 0,C 180,E1 10477.195,E2 10477.195} C_VEL
LIN {X 0,Y 260.042,Z 867.784,A -85,B 0,C 180,E1 10475.015,E2 10475.015} C_VEL
LIN {X 0,Y 267.063,Z 849.969,A -85,B 0,C 180,E1 10473.198,E2 10473.198} C_VEL
LIN {X 0,Y 267.632,Z 848.01,A -85,B 0,C 180,E1 10472.992,E2 10472.992} C_VEL
LIN {X 0,Y 263.101,Z 852.142,A -85,B 0,C 180,E1 10472.273,E2 10472.273} C_VEL
LIN {X 0,Y 255.353,Z 859.406,A -85,B 0,C 180,E1 10471.122,E2 10471.122} C_VEL
LIN {X 0,Y 254.758,Z 859.916,A -85,B 0,C 180,E1 10471.017,E2 10471.017} C_VEL
LIN {X 0,Y 248.915,Z 865.481,A -85,B 0,C 180,E1 10470.162,E2 10470.162} C_VEL
LIN {X 0,Y 237.808,Z 876.547,A -85,B 0,C 180,E1 10468.835,E2 10468.835} C_VEL
LIN {X 0,Y 232.697,Z 880.637,A -85,B 0,C 180,E1 10467.889,E2 10467.889} C_VEL
LIN {X 0,Y 231.317,Z 881.519,A -85,B 0,C 180,E1 10467.537,E2 10467.537} C_VEL
LIN {X 0,Y 223.969,Z 886.308,A -85,B 0,C 180,E1 10465.661,E2 10465.661} C_VEL
LIN {X 0,Y 218.32,Z 889.5,A -85,B 0,C 180,E1 10463.768,E2 10463.768} C_VEL
LIN {X 0,Y 212.688,Z 892.956,A -85,B 0,C 180,E1 10461.801,E2 10461.801} C_VEL
LIN {X 0,Y 209.02,Z 894.806,A -85,B 0,C 180,E1 10460.147,E2 10460.147} C_VEL
LIN {X 0,Y 204.132,Z 897.74,A -85,B 0,C 180,E1 10457.974,E2 10457.974} C_VEL
LIN {X 0,Y 201.142,Z 899.267,A -85,B 0,C 180,E1 10456.163,E2 10456.163} C_VEL
LIN {X 0,Y 197.173,Z 901.77,A -85,B 0,C 180,E1 10453.789,E2 10453.789} C_VEL
LIN {X 0,Y 195.263,Z 902.76,A -85,B 0,C 180,E1 10452.12,E2 10452.12} C_VEL
LIN {X 0,Y 191.965,Z 905.028,A -85,B 0,C 180,E1 10449.595,E2 10449.595} C_VEL
LIN {X 0,Y 190.374,Z 905.987,A -85,B 0,C 180,E1 10447.545,E2 10447.545} C_VEL
LIN {X 0,Y 187.928,Z 908.067,A -85,B 0,C 180,E1 10444.884,E2 10444.884} C_VEL
LIN {X 0,Y 187.221,Z 908.87,A -85,B 0,C 180,E1 10442.755,E2 10442.755} C_VEL
LIN {X 0,Y 187.533,Z 917.249,A -85,B 0,C 180,E1 10437.556,E2 10437.556} C_VEL
LIN {X 0,Y 189.004,Z 924.026,A -85,B 0,C 180,E1 10432.095,E2 10432.095} C_VEL
LIN {X 0,Y 192.224,Z 929.347,A -85,B 0,C 180,E1 10426.157,E2 10426.157} C_VEL
LIN {X 0,Y 197.298,Z 932.55,A -85,B 0,C 180,E1 10420.46,E2 10420.46} C_VEL
LIN {X 0,Y 204.24,Z 933.763,A -85,B 0,C 180,E1 10415.102,E2 10415.102} C_VEL
LIN {X 0,Y 213.009,Z 933.14,A -85,B 0,C 180,E1 10410.162,E2 10410.162} C_VEL
LIN {X 0,Y 223.513,Z 930.776,A -85,B 0,C 180,E1 10405.692,E2 10405.692} C_VEL
LIN {X 0,Y 235.12,Z 926.987,A -85,B 0,C 180,E1 10401.784,E2 10401.784} C_VEL
LIN {X 0,Y 225.248,Z 933.815,A -85,B 0,C 180,E1 10398.932,E2 10398.932} C_VEL
LIN {X 0,Y 216.486,Z 947.313,A -85,B 0,C 180,E1 10395.34,E2 10395.34} C_VEL
LIN {X 0,Y 208.104,Z 959.594,A -85,B 0,C 180,E1 10391.167,E2 10391.167} C_VEL
LIN {X 0,Y 200.536,Z 970.491,A -85,B 0,C 180,E1 10386.395,E2 10386.395} C_VEL
LIN {X 0,Y 194.083,Z 979.926,A -85,B 0,C 180,E1 10381.011,E2 10381.011} C_VEL
LIN {X 0,Y 189.076,Z 987.806,A -85,B 0,C 180,E1 10375.029,E2 10375.029} C_VEL
LIN {X 0,Y 185.934,Z 993.811,A -85,B 0,C 180,E1 10368.825,E2 10368.825} C_VEL
LIN {X 0,Y 184.465,Z 998.064,A -85,B 0,C 180,E1 10362.524,E2 10362.524} C_VEL
LIN {X 0,Y 184.245,Z 1000.561,A -85,B 0,C 180,E1 10356.545,E2 10356.545} C_VEL
LIN {X 0,Y 184.431,Z 1001.423,A -85,B 0,C 180,E1 10351.555,E2 10351.555} C_VEL
LIN {X 0,Y 184.372,Z 1001.293,A -85,B 0,C 180,E1 10346.893,E2 10346.893} C_VEL
LIN {X 0,Y 184.218,Z 999.903,A -85,B 0,C 180,E1 10341.575,E2 10341.575} C_VEL
LIN {X 0,Y 184.717,Z 996.985,A -85,B 0,C 180,E1 10335.584,E2 10335.584} C_VEL
LIN {X 0,Y 186.811,Z 991.92,A -85,B 0,C 180,E1 10328.987,E2 10328.987} C_VEL
LIN {X 0,Y 190.59,Z 985.205,A -85,B 0,C 180,E1 10322.846,E2 10322.846} C_VEL
LIN {X 0,Y 195.887,Z 977.037,A -85,B 0,C 180,E1 10317.247,E2 10317.247} C_VEL
LIN {X 0,Y 202.857,Z 966.955,A -85,B 0,C 180,E1 10311.969,E2 10311.969} C_VEL
LIN {X 0,Y 210.93,Z 955.3,A -85,B 0,C 180,E1 10307.284,E2 10307.284} C_VEL
LIN {X 0,Y 219.651,Z 942.337,A -85,B 0,C 180,E1 10303.256,E2 10303.256} C_VEL
LIN {X 0,Y 228.526,Z 928.294,A -85,B 0,C 180,E1 10299.84,E2 10299.84} C_VEL
LIN {X 0,Y 237.89,Z 912.218,A -85,B 0,C 180,E1 10296.807,E2 10296.807} C_VEL
LIN {X 0,Y 246.876,Z 894.98,A -85,B 0,C 180,E1 10294.291,E2 10294.291} C_VEL
LIN {X 0,Y 254.911,Z 877.417,A -85,B 0,C 180,E1 10292.301,E2 10292.301} C_VEL
LIN {X 0,Y 262.175,Z 859.061,A -85,B 0,C 180,E1 10290.687,E2 10290.687} C_VEL
LIN {X 0,Y 268.553,Z 839.926,A -85,B 0,C 180,E1 10289.402,E2 10289.402} C_VEL
LIN {X 0,Y 273.909,Z 820.007,A -85,B 0,C 180,E1 10288.41,E2 10288.41} C_VEL
LIN {X 0,Y 278.03,Z 799.436,A -85,B 0,C 180,E1 10287.667,E2 10287.667} C_VEL
LIN {X 0,Y 280.734,Z 778.749,A -85,B 0,C 180,E1 10287.153,E2 10287.153} C_VEL
LIN {X 0,Y 284.131,Z 749.221,A -85,B 0,C 180,E1 10286.883,E2 10286.883} C_VEL
LIN {X 0,Y 284.779,Z 743.316,A -85,B 0,C 180,E1 10286.818,E2 10286.818} C_VEL
LIN {X 0,Y 281.316,Z 718.663,A -85,B 0,C 180,E1 10283.944,E2 10283.944} C_VEL
LIN {X 0,Y 279.319,Z 693.935,A -85,B 0,C 180,E1 10281.387,E2 10281.387} C_VEL
LIN {X 0,Y 278.388,Z 668.953,A -85,B 0,C 180,E1 10279.076,E2 10279.076} C_VEL
LIN {X 0,Y 278.272,Z 645.633,A -85,B 0,C 180,E1 10277.135,E2 10277.135} C_VEL
LIN {X 0,Y 273.485,Z 626.415,A -85,B 0,C 180,E1 10271.333,E2 10271.333} C_VEL
LIN {X 0,Y 272.112,Z 619.004,A -85,B 0,C 180,E1 10268.664,E2 10268.664} C_VEL
LIN {X 0,Y 271.007,Z 606.59,A -85,B 0,C 180,E1 10263.754,E2 10263.754} C_VEL
LIN {X 0,Y 271.502,Z 597.22,A -85,B 0,C 180,E1 10259.367,E2 10259.367} C_VEL
LIN {X 0,Y 273.137,Z 590.017,A -85,B 0,C 180,E1 10255.486,E2 10255.486} C_VEL
LIN {X 0,Y 274.448,Z 586.856,A -85,B 0,C 180,E1 10253.41,E2 10253.41} C_VEL
LIN {X 0,Y 277.321,Z 591.875,A -85,B 0,C 180,E1 10248.668,E2 10248.668} C_VEL
LIN {X 0,Y 280.034,Z 596.526,A -85,B 0,C 180,E1 10245.632,E2 10245.632} C_VEL
LIN {X 0,Y 282.904,Z 601.468,A -85,B 0,C 180,E1 10243.047,E2 10243.047} C_VEL
LIN {X 0,Y 286.64,Z 608.08,A -85,B 0,C 180,E1 10240.223,E2 10240.223} C_VEL
LIN {X 0,Y 291.282,Z 616.882,A -85,B 0,C 180,E1 10237.23,E2 10237.23} C_VEL
LIN {X 0,Y 294.179,Z 622.956,A -85,B 0,C 180,E1 10235.548,E2 10235.548} C_VEL
LIN {X 0,Y 281.069,Z 774.131,A -85,B 0,C 180,E1 10232.318,E2 10232.318} C_VEL
LIN {X 0,Y 277.997,Z 794.404,A -85,B 0,C 180,E1 10231.64,E2 10231.64} C_VEL
LIN {X 0,Y 273.568,Z 814.849,A -85,B 0,C 180,E1 10230.675,E2 10230.675} C_VEL
LIN {X 0,Y 268.158,Z 834.045,A -85,B 0,C 180,E1 10229.462,E2 10229.462} C_VEL
LIN {X 0,Y 261.828,Z 852.378,A -85,B 0,C 180,E1 10227.967,E2 10227.967} C_VEL
LIN {X 0,Y 254.253,Z 870.77,A -85,B 0,C 180,E1 10226.053,E2 10226.053} C_VEL
LIN {X 0,Y 245.692,Z 888.545,A -85,B 0,C 180,E1 10223.683,E2 10223.683} C_VEL
LIN {X 0,Y 236.909,Z 904.564,A -85,B 0,C 180,E1 10220.944,E2 10220.944} C_VEL
LIN {X 0,Y 228.074,Z 919.045,A -85,B 0,C 180,E1 10217.805,E2 10217.805} C_VEL
LIN {X 0,Y 219.384,Z 932.108,A -85,B 0,C 180,E1 10214.209,E2 10214.209} C_VEL
LIN {X 0,Y 210.651,Z 944.413,A -85,B 0,C 180,E1 10209.848,E2 10209.848} C_VEL
LIN {X 0,Y 203.091,Z 954.6,A -85,B 0,C 180,E1 10205.169,E2 10205.169} C_VEL
LIN {X 0,Y 196.503,Z 963.366,A -85,B 0,C 180,E1 10199.909,E2 10199.909} C_VEL
LIN {X 0,Y 191.18,Z 970.633,A -85,B 0,C 180,E1 10194.073,E2 10194.073} C_VEL
LIN {X 0,Y 187.366,Z 976.266,A -85,B 0,C 180,E1 10187.707,E2 10187.707} C_VEL
LIN {X 0,Y 185.309,Z 979.878,A -85,B 0,C 180,E1 10181.514,E2 10181.514} C_VEL
LIN {X 0,Y 184.434,Z 981.929,A -85,B 0,C 180,E1 10175.286,E2 10175.286} C_VEL
LIN {X 0,Y 184.283,Z 982.531,A -85,B 0,C 180,E1 10169.687,E2 10169.687} C_VEL
LIN {X 0,Y 184.472,Z 981.831,A -85,B 0,C 180,E1 10164.087,E2 10164.087} C_VEL
LIN {X 0,Y 185.429,Z 979.644,A -85,B 0,C 180,E1 10157.859,E2 10157.859} C_VEL
LIN {X 0,Y 187.616,Z 975.885,A -85,B 0,C 180,E1 10151.672,E2 10151.672} C_VEL
LIN {X 0,Y 191.352,Z 970.445,A -85,B 0,C 180,E1 10145.618,E2 10145.618} C_VEL
LIN {X 0,Y 196.812,Z 963.055,A -85,B 0,C 180,E1 10139.729,E2 10139.729} C_VEL
LIN {X 0,Y 203.392,Z 954.313,A -85,B 0,C 180,E1 10134.542,E2 10134.542} C_VEL
LIN {X 0,Y 211.011,Z 944.055,A -85,B 0,C 180,E1 10129.876,E2 10129.876} C_VEL
LIN {X 0,Y 219.522,Z 932.068,A -85,B 0,C 180,E1 10125.651,E2 10125.651} C_VEL
LIN {X 0,Y 228.53,Z 918.515,A -85,B 0,C 180,E1 10121.944,E2 10121.944} C_VEL
LIN {X 0,Y 237.401,Z 903.925,A -85,B 0,C 180,E1 10118.814,E2 10118.814} C_VEL
LIN {X 0,Y 245.895,Z 888.422,A -85,B 0,C 180,E1 10116.18,E2 10116.18} C_VEL
LIN {X 0,Y 254.163,Z 871.285,A -85,B 0,C 180,E1 10113.893,E2 10113.893} C_VEL
LIN {X 0,Y 257.885,Z 862.443,A -85,B 0,C 180,E1 10112.875,E2 10112.875} C_VEL
LIN {X 0,Y 249.884,Z 868.687,A -85,B 0,C 180,E1 10111.538,E2 10111.538} C_VEL
LIN {X 0,Y 245.1,Z 872.119,A -85,B 0,C 180,E1 10110.596,E2 10110.596} C_VEL
LIN {X 0,Y 237.003,Z 878.03,A -85,B 0,C 180,E1 10109.023,E2 10109.023} C_VEL
LIN {X 0,Y 231.317,Z 881.519,A -85,B 0,C 180,E1 10107.537,E2 10107.537} C_VEL
LIN {X 0,Y 227.844,Z 884.12,A -85,B 0,C 180,E1 10106.812,E2 10106.812} C_VEL
LIN {X 0,Y 217.814,Z 893.395,A -85,B 0,C 180,E1 10105.553,E2 10105.553} C_VEL
LIN {X 0,Y 214.802,Z 895.541,A -85,B 0,C 180,E1 10104.882,E2 10104.882} C_VEL
LIN {X 0,Y 208.811,Z 898.9,A -85,B 0,C 180,E1 10102.822,E2 10102.822} C_VEL
LIN {X 0,Y 204.95,Z 900.859,A -85,B 0,C 180,E1 10101.163,E2 10101.163} C_VEL
LIN {X 0,Y 199.468,Z 903.82,A -85,B 0,C 180,E1 10098.712,E2 10098.712} C_VEL
LIN {X 0,Y 196.703,Z 905.164,A -85,B 0,C 180,E1 10097.128,E2 10097.128} C_VEL
LIN {X 0,Y 192.237,Z 907.675,A -85,B 0,C 180,E1 10094.458,E2 10094.458} C_VEL
LIN {X 0,Y 190.523,Z 908.521,A -85,B 0,C 180,E1 10093.042,E2 10093.042} C_VEL
LIN {X 0,Y 186.846,Z 910.893,A -85,B 0,C 180,E1 10090.172,E2 10090.172} C_VEL
LIN {X 0,Y 185.411,Z 911.715,A -85,B 0,C 180,E1 10088.373,E2 10088.373} C_VEL
LIN {X 0,Y 182.616,Z 913.871,A -85,B 0,C 180,E1 10085.341,E2 10085.341} C_VEL
LIN {X 0,Y 181.62,Z 914.704,A -85,B 0,C 180,E1 10083.156,E2 10083.156} C_VEL
LIN {X 0,Y 179.728,Z 916.891,A -85,B 0,C 180,E1 10079.682,E2 10079.682} C_VEL
LIN {X 0,Y 179.599,Z 917.983,A -85,B 0,C 180,E1 10077.129,E2 10077.129} C_VEL
LIN {X 0,Y 181.227,Z 924.965,A -85,B 0,C 180,E1 10071.434,E2 10071.434} C_VEL
LIN {X 0,Y 184.297,Z 930.11,A -85,B 0,C 180,E1 10065.87,E2 10065.87} C_VEL
LIN {X 0,Y 189.262,Z 933.709,A -85,B 0,C 180,E1 10060.239,E2 10060.239} C_VEL
LIN {X 0,Y 196.798,Z 935.601,A -85,B 0,C 180,E1 10054.415,E2 10054.415} C_VEL
LIN {X 0,Y 206.415,Z 935.504,A -85,B 0,C 180,E1 10049.106,E2 10049.106} C_VEL
LIN {X 0,Y 217.973,Z 933.535,A -85,B 0,C 180,E1 10044.37,E2 10044.37} C_VEL
LIN {X 0,Y 225.053,Z 931.74,A -85,B 0,C 180,E1 10041.953,E2 10041.953} C_VEL
LIN {X 0,Y 218.248,Z 936.052,A -85,B 0,C 180,E1 10039.916,E2 10039.916} C_VEL
LIN {X 0,Y 208.623,Z 950.019,A -85,B 0,C 180,E1 10035.966,E2 10035.966} C_VEL
LIN {X 0,Y 200.074,Z 961.759,A -85,B 0,C 180,E1 10031.658,E2 10031.658} C_VEL
LIN {X 0,Y 192.366,Z 972.173,A -85,B 0,C 180,E1 10026.71,E2 10026.71} C_VEL
LIN {X 0,Y 185.535,Z 981.608,A -85,B 0,C 180,E1 10020.796,E2 10020.796} C_VEL
LIN {X 0,Y 180.61,Z 989.04,A -85,B 0,C 180,E1 10014.534,E2 10014.534} C_VEL
LIN {X 0,Y 177.617,Z 994.647,A -85,B 0,C 180,E1 10008.038,E2 10008.038} C_VEL
LIN {X 0,Y 176.353,Z 998.488,A -85,B 0,C 180,E1 10001.447,E2 10001.447} C_VEL
LIN {X 0,Y 176.287,Z 1000.442,A -85,B 0,C 180,E1 9995.535,E2 9995.535} C_VEL
LIN {X 0,Y 176.465,Z 1001.107,A -85,B 0,C 180,E1 9990.326,E2 9990.326} C_VEL
LIN {X 0,Y 176.303,Z 1000.578,A -85,B 0,C 180,E1 9985.122,E2 9985.122} C_VEL
LIN {X 0,Y 176.292,Z 998.757,A -85,B 0,C 180,E1 9979.214,E2 9979.214} C_VEL
LIN {X 0,Y 177.393,Z 995.05,A -85,B 0,C 180,E1 9972.621,E2 9972.621} C_VEL
LIN {X 0,Y 180.193,Z 989.627,A -85,B 0,C 180,E1 9966.107,E2 9966.107} C_VEL
LIN {X 0,Y 185.196,Z 981.964,A -85,B 0,C 180,E1 9959.504,E2 9959.504} C_VEL
LIN {X 0,Y 191.932,Z 972.616,A -85,B 0,C 180,E1 9953.569,E2 9953.569} C_VEL
LIN {X 0,Y 199.561,Z 962.301,A -85,B 0,C 180,E1 9948.598,E2 9948.598} C_VEL
LIN {X 0,Y 208.034,Z 950.67,A -85,B 0,C 180,E1 9944.266,E2 9944.266} C_VEL
LIN {X 0,Y 217.599,Z 936.789,A -85,B 0,C 180,E1 9940.294,E2 9940.294} C_VEL
LIN {X 0,Y 227.181,Z 921.747,A -85,B 0,C 180,E1 9936.986,E2 9936.986} C_VEL
LIN {X 0,Y 236.131,Z 906.31,A -85,B 0,C 180,E1 9934.343,E2 9934.343} C_VEL
LIN {X 0,Y 245.133,Z 888.937,A -85,B 0,C 180,E1 9932.022,E2 9932.022} C_VEL
LIN {X 0,Y 253.627,Z 870.068,A -85,B 0,C 180,E1 9930.083,E2 9930.083} C_VEL
LIN {X 0,Y 260.819,Z 851.306,A -85,B 0,C 180,E1 9928.615,E2 9928.615} C_VEL
LIN {X 0,Y 267.047,Z 831.662,A -85,B 0,C 180,E1 9927.459,E2 9927.459} C_VEL
LIN {X 0,Y 272.156,Z 811.041,A -85,B 0,C 180,E1 9926.577,E2 9926.577} C_VEL
LIN {X 0,Y 275.861,Z 789.354,A -85,B 0,C 180,E1 9925.903,E2 9925.903} C_VEL
LIN {X 0,Y 278.628,Z 765.065,A -85,B 0,C 180,E1 9925.52,E2 9925.52} C_VEL
LIN {X 0,Y 280.963,Z 745.311,A -85,B 0,C 180,E1 9925.37,E2 9925.37} C_VEL
LIN {X 0,Y 277.97,Z 721.366,A -85,B 0,C 180,E1 9922.538,E2 9922.538} C_VEL
LIN {X 0,Y 276.325,Z 696.865,A -85,B 0,C 180,E1 9919.981,E2 9919.981} C_VEL
LIN {X 0,Y 275.672,Z 672.044,A -85,B 0,C 180,E1 9917.656,E2 9917.656} C_VEL
LIN {X 0,Y 275.745,Z 650.59,A -85,B 0,C 180,E1 9915.834,E2 9915.834} C_VEL
LIN {X 0,Y 271.541,Z 631.222,A -85,B 0,C 180,E1 9909.858,E2 9909.858} C_VEL
LIN {X 0,Y 269.91,Z 613.73,A -85,B 0,C 180,E1 9903.026,E2 9903.026} C_VEL
LIN {X 0,Y 270.67,Z 604.377,A -85,B 0,C 180,E1 9898.624,E2 9898.624} C_VEL
LIN {X 0,Y 272.539,Z 597.222,A -85,B 0,C 180,E1 9894.737,E2 9894.737} C_VEL
LIN {X 0,Y 273.445,Z 595.071,A -85,B 0,C 180,E1 9893.386,E2 9893.386} C_VEL
LIN {X 0,Y 276.022,Z 599.595,A -85,B 0,C 180,E1 9889.026,E2 9889.026} C_VEL
LIN {X 0,Y 278.534,Z 604.077,A -85,B 0,C 180,E1 9886.083,E2 9886.083} C_VEL
LIN {X 0,Y 281.42,Z 609.244,A -85,B 0,C 180,E1 9883.38,E2 9883.38} C_VEL
LIN {X 0,Y 285.609,Z 616.995,A -85,B 0,C 180,E1 9880.149,E2 9880.149} C_VEL
LIN {X 0,Y 290.364,Z 626.68,A -85,B 0,C 180,E1 9877.047,E2 9877.047} C_VEL
LIN {X 0,Y 290.573,Z 627.55,A -85,B 0,C 180,E1 9876.894,E2 9876.894} C_VEL
LIN {X 0,Y 277.434,Z 774.562,A -85,B 0,C 180,E1 9873.777,E2 9873.777} C_VEL
LIN {X 0,Y 274.263,Z 794.909,A -85,B 0,C 180,E1 9873.105,E2 9873.105} C_VEL
LIN {X 0,Y 269.728,Z 815.272,A -85,B 0,C 180,E1 9872.155,E2 9872.155} C_VEL
LIN {X 0,Y 264.177,Z 834.437,A -85,B 0,C 180,E1 9870.959,E2 9870.959} C_VEL
LIN {X 0,Y 257.662,Z 852.777,A -85,B 0,C 180,E1 9869.48,E2 9869.48} C_VEL
LIN {X 0,Y 249.888,Z 871.102,A -85,B 0,C 180,E1 9867.591,E2 9867.591} C_VEL
LIN {X 0,Y 241.341,Z 888.3,A -85,B 0,C 180,E1 9865.321,E2 9865.321} C_VEL
LIN {X 0,Y 232.412,Z 904.106,A -85,B 0,C 180,E1 9862.656,E2 9862.656} C_VEL
LIN {X 0,Y 223.314,Z 918.553,A -85,B 0,C 180,E1 9859.564,E2 9859.564} C_VEL
LIN {X 0,Y 214.034,Z 931.997,A -85,B 0,C 180,E1 9855.888,E2 9855.888} C_VEL
LIN {X 0,Y 204.967,Z 944.211,A -85,B 0,C 180,E1 9851.56,E2 9851.56} C_VEL
LIN {X 0,Y 196.917,Z 954.518,A -85,B 0,C 180,E1 9846.807,E2 9846.807} C_VEL
LIN {X 0,Y 189.838,Z 963.392,A -85,B 0,C 180,E1 9841.426,E2 9841.426} C_VEL
LIN {X 0,Y 183.804,Z 971.051,A -85,B 0,C 180,E1 9835.105,E2 9835.105} C_VEL
LIN {X 0,Y 179.679,Z 976.683,A -85,B 0,C 180,E1 9828.491,E2 9828.491} C_VEL
LIN {X 0,Y 177.423,Z 980.293,A -85,B 0,C 180,E1 9822.033,E2 9822.033} C_VEL
LIN {X 0,Y 176.484,Z 982.278,A -85,B 0,C 180,E1 9815.851,E2 9815.851} C_VEL
LIN {X 0,Y 176.3,Z 982.952,A -85,B 0,C 180,E1 9809.998,E2 9809.998} C_VEL
LIN {X 0,Y 176.478,Z 982.307,A -85,B 0,C 180,E1 9804.145,E2 9804.145} C_VEL
LIN {X 0,Y 177.48,Z 980.21,A -85,B 0,C 180,E1 9797.637,E2 9797.637} C_VEL
LIN {X 0,Y 179.796,Z 976.544,A -85,B 0,C 180,E1 9791.182,E2 9791.182} C_VEL
LIN {X 0,Y 183.749,Z 971.176,A -85,B 0,C 180,E1 9784.883,E2 9784.883} C_VEL
LIN {X 0,Y 189.434,Z 963.948,A -85,B 0,C 180,E1 9778.85,E2 9778.85} C_VEL
LIN {X 0,Y 196.42,Z 955.227,A -85,B 0,C 180,E1 9773.444,E2 9773.444} C_VEL
LIN {X 0,Y 204.392,Z 945.086,A -85,B 0,C 180,E1 9768.667,E2 9768.667} C_VEL
LIN {X 0,Y 213.576,Z 932.792,A -85,B 0,C 180,E1 9764.231,E2 9764.231} C_VEL
LIN {X 0,Y 222.613,Z 919.827,A -85,B 0,C 180,E1 9760.617,E2 9760.617} C_VEL
LIN {X 0,Y 231.836,Z 905.344,A -85,B 0,C 180,E1 9757.453,E2 9757.453} C_VEL
LIN {X 0,Y 240.893,Z 889.455,A -85,B 0,C 180,E1 9754.73,E2 9754.73} C_VEL
LIN {X 0,Y 248.305,Z 874.679,A -85,B 0,C 180,E1 9752.724,E2 9752.724} C_VEL
LIN {X 0,Y 243.876,Z 877.728,A -85,B 0,C 180,E1 9751.931,E2 9751.931} C_VEL
LIN {X 0,Y 235.079,Z 883.79,A -85,B 0,C 180,E1 9750.295,E2 9750.295} C_VEL
LIN {X 0,Y 227.527,Z 888.254,A -85,B 0,C 180,E1 9748.488,E2 9748.488} C_VEL
LIN {X 0,Y 220.391,Z 892.57,A -85,B 0,C 180,E1 9746.65,E2 9746.65} C_VEL
LIN {X 0,Y 215.063,Z 895.384,A -85,B 0,C 180,E1 9744.959,E2 9744.959} C_VEL
LIN {X 0,Y 214.802,Z 895.541,A -85,B 0,C 180,E1 9744.882,E2 9744.882} C_VEL
LIN {X 0,Y 207.052,Z 900.834,A -85,B 0,C 180,E1 9742.791,E2 9742.791} C_VEL
LIN {X 0,Y 197.111,Z 907.885,A -85,B 0,C 180,E1 9740.086,E2 9740.086} C_VEL
LIN {X 0,Y 192.751,Z 910.597,A -85,B 0,C 180,E1 9738.407,E2 9738.407} C_VEL
LIN {X 0,Y 187.565,Z 913.267,A -85,B 0,C 180,E1 9735.459,E2 9735.459} C_VEL
LIN {X 0,Y 185.252,Z 914.401,A -85,B 0,C 180,E1 9733.738,E2 9733.738} C_VEL
LIN {X 0,Y 181.533,Z 916.544,A -85,B 0,C 180,E1 9730.794,E2 9730.794} C_VEL
LIN {X 0,Y 179.892,Z 917.47,A -85,B 0,C 180,E1 9728.954,E2 9728.954} C_VEL
LIN {X 0,Y 176.935,Z 919.617,A -85,B 0,C 180,E1 9725.513,E2 9725.513} C_VEL
LIN {X 0,Y 175.964,Z 920.418,A -85,B 0,C 180,E1 9723.584,E2 9723.584} C_VEL
LIN {X 0,Y 173.979,Z 922.582,A -85,B 0,C 180,E1 9719.671,E2 9719.671} C_VEL
LIN {X 0,Y 173.513,Z 923.634,A -85,B 0,C 180,E1 9717.028,E2 9717.028} C_VEL
LIN {X 0,Y 173.168,Z 926.044,A -85,B 0,C 180,E1 9712.035,E2 9712.035} C_VEL
LIN {X 0,Y 173.914,Z 926.886,A -85,B 0,C 180,E1 9709.734,E2 9709.734} C_VEL
LIN {X 0,Y 177.537,Z 931.984,A -85,B 0,C 180,E1 9703.981,E2 9703.981} C_VEL
LIN {X 0,Y 183.182,Z 935.601,A -85,B 0,C 180,E1 9698.213,E2 9698.213} C_VEL
LIN {X 0,Y 191.545,Z 937.578,A -85,B 0,C 180,E1 9692.318,E2 9692.318} C_VEL
LIN {X 0,Y 202.017,Z 937.629,A -85,B 0,C 180,E1 9687.015,E2 9687.015} C_VEL
LIN {X 0,Y 215.016,Z 935.777,A -85,B 0,C 180,E1 9682.134,E2 9682.134} C_VEL
LIN {X 0,Y 211.513,Z 937.79,A -85,B 0,C 180,E1 9681.045,E2 9681.045} C_VEL
LIN {X 0,Y 201.88,Z 951.102,A -85,B 0,C 180,E1 9677.141,E2 9677.141} C_VEL
LIN {X 0,Y 192.537,Z 963.273,A -85,B 0,C 180,E1 9672.464,E2 9672.464} C_VEL
LIN {X 0,Y 184.204,Z 973.856,A -85,B 0,C 180,E1 9667.052,E2 9667.052} C_VEL
LIN {X 0,Y 177.469,Z 982.581,A -85,B 0,C 180,E1 9661.09,E2 9661.09} C_VEL
LIN {X 0,Y 172.536,Z 989.562,A -85,B 0,C 180,E1 9654.663,E2 9654.663} C_VEL
LIN {X 0,Y 169.418,Z 995.094,A -85,B 0,C 180,E1 9647.519,E2 9647.519} C_VEL
LIN {X 0,Y 168.297,Z 998.602,A -85,B 0,C 180,E1 9640.615,E2 9640.615} C_VEL
LIN {X 0,Y 168.318,Z 1000.248,A -85,B 0,C 180,E1 9634.772,E2 9634.772} C_VEL
LIN {X 0,Y 168.475,Z 1000.692,A -85,B 0,C 180,E1 9629.662,E2 9629.662} C_VEL
LIN {X 0,Y 168.29,Z 1000.091,A -85,B 0,C 180,E1 9624.547,E2 9624.547} C_VEL
LIN {X 0,Y 168.354,Z 998.208,A -85,B 0,C 180,E1 9618.352,E2 9618.352} C_VEL
LIN {X 0,Y 169.716,Z 994.411,A -85,B 0,C 180,E1 9611.452,E2 9611.452} C_VEL
LIN {X 0,Y 172.916,Z 988.889,A -85,B 0,C 180,E1 9604.668,E2 9604.668} C_VEL
LIN {X 0,Y 178.14,Z 981.539,A -85,B 0,C 180,E1 9598.159,E2 9598.159} C_VEL
LIN {X 0,Y 185.362,Z 972.192,A -85,B 0,C 180,E1 9592.055,E2 9592.055} C_VEL
LIN {X 0,Y 193.459,Z 961.878,A -85,B 0,C 180,E1 9586.985,E2 9586.985} C_VEL
LIN {X 0,Y 202.387,Z 950.238,A -85,B 0,C 180,E1 9582.596,E2 9582.596} C_VEL
LIN {X 0,Y 212.389,Z 936.37,A -85,B 0,C 180,E1 9578.606,E2 9578.606} C_VEL
LIN {X 0,Y 222.36,Z 921.331,A -85,B 0,C 180,E1 9575.303,E2 9575.303} C_VEL
LIN {X 0,Y 231.864,Z 905.495,A -85,B 0,C 180,E1 9572.617,E2 9572.617} C_VEL
LIN {X 0,Y 241.022,Z 888.338,A -85,B 0,C 180,E1 9570.362,E2 9570.362} C_VEL
LIN {X 0,Y 249.709,Z 869.576,A -85,B 0,C 180,E1 9568.469,E2 9568.469} C_VEL
LIN {X 0,Y 257.054,Z 850.912,A -85,B 0,C 180,E1 9567.037,E2 9567.037} C_VEL
LIN {X 0,Y 263.435,Z 831.279,A -85,B 0,C 180,E1 9565.907,E2 9565.907} C_VEL
LIN {X 0,Y 268.658,Z 810.674,A -85,B 0,C 180,E1 9565.045,E2 9565.045} C_VEL
LIN {X 0,Y 272.474,Z 788.831,A -85,B 0,C 180,E1 9564.379,E2 9564.379} C_VEL
LIN {X 0,Y 275.376,Z 763.909,A -85,B 0,C 180,E1 9564.01,E2 9564.01} C_VEL
LIN {X 0,Y 277.342,Z 747.375,A -85,B 0,C 180,E1 9563.892,E2 9563.892} C_VEL
LIN {X 0,Y 274.789,Z 723.94,A -85,B 0,C 180,E1 9561.086,E2 9561.086} C_VEL
LIN {X 0,Y 273.376,Z 696.736,A -85,B 0,C 180,E1 9558.222,E2 9558.222} C_VEL
LIN {X 0,Y 273.192,Z 667.411,A -85,B 0,C 180,E1 9555.537,E2 9555.537} C_VEL
LIN {X 0,Y 273.409,Z 655.703,A -85,B 0,C 180,E1 9554.561,E2 9554.561} C_VEL
LIN {X 0,Y 269.829,Z 636.546,A -85,B 0,C 180,E1 9548.523,E2 9548.523} C_VEL
LIN {X 0,Y 268.863,Z 620.64,A -85,B 0,C 180,E1 9542.184,E2 9542.184} C_VEL
LIN {X 0,Y 269.904,Z 611.429,A -85,B 0,C 180,E1 9537.824,E2 9537.824} C_VEL
LIN {X 0,Y 272.06,Z 604.245,A -85,B 0,C 180,E1 9533.881,E2 9533.881} C_VEL
LIN {X 0,Y 272.493,Z 603.337,A -85,B 0,C 180,E1 9533.257,E2 9533.257} C_VEL
LIN {X 0,Y 274.72,Z 607.282,A -85,B 0,C 180,E1 9529.409,E2 9529.409} C_VEL
LIN {X 0,Y 277.145,Z 611.811,A -85,B 0,C 180,E1 9526.437,E2 9526.437} C_VEL
LIN {X 0,Y 280.472,Z 617.9,A -85,B 0,C 180,E1 9523.269,E2 9523.269} C_VEL
LIN {X 0,Y 285.112,Z 627.175,A -85,B 0,C 180,E1 9519.685,E2 9519.685} C_VEL
LIN {X 0,Y 287.155,Z 631.886,A -85,B 0,C 180,E1 9518.279,E2 9518.279} C_VEL
LIN {X 0,Y 273.983,Z 774.99,A -85,B 0,C 180,E1 9515.275,E2 9515.275} C_VEL
LIN {X 0,Y 270.74,Z 795.274,A -85,B 0,C 180,E1 9514.614,E2 9514.614} C_VEL
LIN {X 0,Y 266.071,Z 815.705,A -85,B 0,C 180,E1 9513.677,E2 9513.677} C_VEL
LIN {X 0,Y 260.382,Z 834.83,A -85,B 0,C 180,E1 9512.5,E2 9512.5} C_VEL
LIN {X 0,Y 253.681,Z 853.176,A -85,B 0,C 180,E1 9511.041,E2 9511.041} C_VEL
LIN {X 0,Y 245.674,Z 871.505,A -85,B 0,C 180,E1 9509.173,E2 9509.173} C_VEL
LIN {X 0,Y 236.852,Z 888.707,A -85,B 0,C 180,E1 9506.923,E2 9506.923} C_VEL
LIN {X 0,Y 227.43,Z 904.809,A -85,B 0,C 180,E1 9504.217,E2 9504.217} C_VEL
LIN {X 0,Y 218.156,Z 918.966,A -85,B 0,C 180,E1 9501.181,E2 9501.181} C_VEL
LIN {X 0,Y 208.251,Z 932.712,A -85,B 0,C 180,E1 9497.392,E2 9497.392} C_VEL
LIN {X 0,Y 198.967,Z 944.628,A -85,B 0,C 180,E1 9493.111,E2 9493.111} C_VEL
LIN {X 0,Y 190.477,Z 954.936,A -85,B 0,C 180,E1 9488.271,E2 9488.271} C_VEL
LIN {X 0,Y 182.777,Z 964.008,A -85,B 0,C 180,E1 9482.601,E2 9482.601} C_VEL
LIN {X 0,Y 176.491,Z 971.469,A -85,B 0,C 180,E1 9476.222,E2 9476.222} C_VEL
LIN {X 0,Y 172.027,Z 977.1,A -85,B 0,C 180,E1 9469.346,E2 9469.346} C_VEL
LIN {X 0,Y 169.55,Z 980.708,A -85,B 0,C 180,E1 9462.601,E2 9462.601} C_VEL
LIN {X 0,Y 168.515,Z 982.69,A -85,B 0,C 180,E1 9456.129,E2 9456.129} C_VEL
LIN {X 0,Y 168.31,Z 983.364,A -85,B 0,C 180,E1 9449.998,E2 9449.998} C_VEL
LIN {X 0,Y 168.509,Z 982.719,A -85,B 0,C 180,E1 9443.867,E2 9443.867} C_VEL
LIN {X 0,Y 169.615,Z 980.624,A -85,B 0,C 180,E1 9437.054,E2 9437.054} C_VEL
LIN {X 0,Y 172.157,Z 976.96,A -85,B 0,C 180,E1 9430.313,E2 9430.313} C_VEL
LIN {X 0,Y 176.697,Z 971.276,A -85,B 0,C 180,E1 9423.445,E2 9423.445} C_VEL
LIN {X 0,Y 182.883,Z 963.972,A -85,B 0,C 180,E1 9417.229,E2 9417.229} C_VEL
LIN {X 0,Y 190.39,Z 955.142,A -85,B 0,C 180,E1 9411.704,E2 9411.704} C_VEL
LIN {X 0,Y 198.871,Z 944.88,A -85,B 0,C 180,E1 9406.859,E2 9406.859} C_VEL
LIN {X 0,Y 207.976,Z 933.241,A -85,B 0,C 180,E1 9402.643,E2 9402.643} C_VEL
LIN {X 0,Y 217.433,Z 920.234,A -85,B 0,C 180,E1 9398.998,E2 9398.998} C_VEL
LIN {X 0,Y 226.974,Z 905.818,A -85,B 0,C 180,E1 9395.848,E2 9395.848} C_VEL
LIN {X 0,Y 236.396,Z 889.854,A -85,B 0,C 180,E1 9393.125,E2 9393.125} C_VEL
LIN {X 0,Y 238.224,Z 886.244,A -85,B 0,C 180,E1 9392.57,E2 9392.57} C_VEL
LIN {X 0,Y 229.861,Z 891.267,A -85,B 0,C 180,E1 9390.883,E2 9390.883} C_VEL
LIN {X 0,Y 224.344,Z 894.379,A -85,B 0,C 180,E1 9389.646,E2 9389.646} C_VEL
LIN {X 0,Y 216.208,Z 898.876,A -85,B 0,C 180,E1 9387.546,E2 9387.546} C_VEL
LIN {X 0,Y 212.141,Z 900.935,A -85,B 0,C 180,E1 9386.298,E2 9386.298} C_VEL
LIN {X 0,Y 205.438,Z 904.407,A -85,B 0,C 180,E1 9384.132,E2 9384.132} C_VEL
LIN {X 0,Y 200.739,Z 906.661,A -85,B 0,C 180,E1 9382.244,E2 9382.244} C_VEL
LIN {X 0,Y 194.693,Z 909.716,A -85,B 0,C 180,E1 9379.501,E2 9379.501} C_VEL
LIN {X 0,Y 192.751,Z 910.597,A -85,B 0,C 180,E1 9378.407,E2 9378.407} C_VEL
LIN {X 0,Y 186.688,Z 914.446,A -85,B 0,C 180,E1 9375.863,E2 9375.863} C_VEL
LIN {X 0,Y 177.243,Z 921.091,A -85,B 0,C 180,E1 9371.64,E2 9371.64} C_VEL
LIN {X 0,Y 174.508,Z 922.882,A -85,B 0,C 180,E1 9369.777,E2 9369.777} C_VEL
LIN {X 0,Y 171.243,Z 925.012,A -85,B 0,C 180,E1 9366.033,E2 9366.033} C_VEL
LIN {X 0,Y 170.118,Z 925.866,A -85,B 0,C 180,E1 9364.045,E2 9364.045} C_VEL
LIN {X 0,Y 168.037,Z 928.049,A -85,B 0,C 180,E1 9359.66,E2 9359.66} C_VEL
LIN {X 0,Y 167.672,Z 928.82,A -85,B 0,C 180,E1 9357.608,E2 9357.608} C_VEL
LIN {X 0,Y 167.106,Z 931.215,A -85,B 0,C 180,E1 9352.437,E2 9352.437} C_VEL
LIN {X 0,Y 167.871,Z 932.441,A -85,B 0,C 180,E1 9349.013,E2 9349.013} C_VEL
LIN {X 0,Y 170.976,Z 935.059,A -85,B 0,C 180,E1 9342.297,E2 9342.297} C_VEL
LIN {X 0,Y 175.859,Z 936.841,A -85,B 0,C 180,E1 9337.256,E2 9337.256} C_VEL
LIN {X 0,Y 184.191,Z 939.231,A -85,B 0,C 180,E1 9331.466,E2 9331.466} C_VEL
LIN {X 0,Y 195.053,Z 939.889,A -85,B 0,C 180,E1 9326.032,E2 9326.032} C_VEL
LIN {X 0,Y 204.867,Z 939.513,A -85,B 0,C 180,E1 9322.248,E2 9322.248} C_VEL
LIN {X 0,Y 194.422,Z 953.102,A -85,B 0,C 180,E1 9318.045,E2 9318.045} C_VEL
LIN {X 0,Y 185.033,Z 964.616,A -85,B 0,C 180,E1 9313.338,E2 9313.338} C_VEL
LIN {X 0,Y 176.857,Z 974.433,A -85,B 0,C 180,E1 9308.044,E2 9308.044} C_VEL
LIN {X 0,Y 169.624,Z 983.253,A -85,B 0,C 180,E1 9301.644,E2 9301.644} C_VEL
LIN {X 0,Y 164.263,Z 990.398,A -85,B 0,C 180,E1 9294.453,E2 9294.453} C_VEL
LIN {X 0,Y 161.325,Z 995.325,A -85,B 0,C 180,E1 9287.309,E2 9287.309} C_VEL
LIN {X 0,Y 160.289,Z 998.428,A -85,B 0,C 180,E1 9280.424,E2 9280.424} C_VEL
LIN {X 0,Y 160.345,Z 999.98,A -85,B 0,C 180,E1 9274.293,E2 9274.293} C_VEL
LIN {X 0,Y 160.471,Z 1000.233,A -85,B 0,C 180,E1 9268.931,E2 9268.931} C_VEL
LIN {X 0,Y 160.256,Z 999.528,A -85,B 0,C 180,E1 9263.554,E2 9263.554} C_VEL
LIN {X 0,Y 160.526,Z 997.288,A -85,B 0,C 180,E1 9256.678,E2 9256.678} C_VEL
LIN {X 0,Y 162.418,Z 993.222,A -85,B 0,C 180,E1 9249.344,E2 9249.344} C_VEL
LIN {X 0,Y 166.595,Z 987.05,A -85,B 0,C 180,E1 9241.914,E2 9241.914} C_VEL
LIN {X 0,Y 172.933,Z 979.031,A -85,B 0,C 180,E1 9235.085,E2 9235.085} C_VEL
LIN {X 0,Y 180.716,Z 969.665,A -85,B 0,C 180,E1 9229.244,E2 9229.244} C_VEL
LIN {X 0,Y 189.618,Z 958.871,A -85,B 0,C 180,E1 9224.184,E2 9224.184} C_VEL
LIN {X 0,Y 199.278,Z 946.707,A -85,B 0,C 180,E1 9219.858,E2 9219.858} C_VEL
LIN {X 0,Y 209.313,Z 933.18,A -85,B 0,C 180,E1 9216.171,E2 9216.171} C_VEL
LIN {X 0,Y 219.131,Z 918.805,A -85,B 0,C 180,E1 9213.149,E2 9213.149} C_VEL
LIN {X 0,Y 229.03,Z 902.667,A -85,B 0,C 180,E1 9210.532,E2 9210.532} C_VEL
LIN {X 0,Y 238.174,Z 885.716,A -85,B 0,C 180,E1 9208.42,E2 9208.42} C_VEL
LIN {X 0,Y 246.311,Z 868.366,A -85,B 0,C 180,E1 9206.743,E2 9206.743} C_VEL
LIN {X 0,Y 253.896,Z 849.395,A -85,B 0,C 180,E1 9205.342,E2 9205.342} C_VEL
LIN {X 0,Y 260.294,Z 829.925,A -85,B 0,C 180,E1 9204.268,E2 9204.268} C_VEL
LIN {X 0,Y 265.459,Z 809.794,A -85,B 0,C 180,E1 9203.456,E2 9203.456} C_VEL
LIN {X 0,Y 269.289,Z 788.287,A -85,B 0,C 180,E1 9202.819,E2 9202.819} C_VEL
LIN {X 0,Y 272.299,Z 762.936,A -85,B 0,C 180,E1 9202.467,E2 9202.467} C_VEL
LIN {X 0,Y 273.888,Z 749.511,A -85,B 0,C 180,E1 9202.369,E2 9202.369} C_VEL
LIN {X 0,Y 271.594,Z 723.106,A -85,B 0,C 180,E1 9199.223,E2 9199.223} C_VEL
LIN {X 0,Y 270.701,Z 695.311,A -85,B 0,C 180,E1 9196.316,E2 9196.316} C_VEL
LIN {X 0,Y 271.057,Z 665.055,A -85,B 0,C 180,E1 9193.601,E2 9193.601} C_VEL
LIN {X 0,Y 271.166,Z 660.679,A -85,B 0,C 180,E1 9193.215,E2 9193.215} C_VEL
LIN {X 0,Y 268.342,Z 642.864,A -85,B 0,C 180,E1 9187.493,E2 9187.493} C_VEL
LIN {X 0,Y 267.868,Z 627.664,A -85,B 0,C 180,E1 9181.39,E2 9181.39} C_VEL
LIN {X 0,Y 269.167,Z 618.581,A -85,B 0,C 180,E1 9177.072,E2 9177.072} C_VEL
LIN {X 0,Y 271.521,Z 611.547,A -85,B 0,C 180,E1 9173.179,E2 9173.179} C_VEL
LIN {X 0,Y 273.438,Z 614.984,A -85,B 0,C 180,E1 9169.784,E2 9169.784} C_VEL
LIN {X 0,Y 275.767,Z 619.542,A -85,B 0,C 180,E1 9166.795,E2 9166.795} C_VEL
LIN {X 0,Y 278.818,Z 625.409,A -85,B 0,C 180,E1 9163.757,E2 9163.757} C_VEL
LIN {X 0,Y 283.1,Z 634.362,A -85,B 0,C 180,E1 9160.288,E2 9160.288} C_VEL
LIN {X 0,Y 283.898,Z 636.311,A -85,B 0,C 180,E1 9159.695,E2 9159.695} C_VEL
LIN {X 0,Y 270.713,Z 775.524,A -85,B 0,C 180,E1 9156.807,E2 9156.807} C_VEL
LIN {X 0,Y 267.382,Z 795.777,A -85,B 0,C 180,E1 9156.158,E2 9156.158} C_VEL
LIN {X 0,Y 262.609,Z 816.127,A -85,B 0,C 180,E1 9155.24,E2 9155.24} C_VEL
LIN {X 0,Y 256.78,Z 835.222,A -85,B 0,C 180,E1 9154.086,E2 9154.086} C_VEL
LIN {X 0,Y 249.896,Z 853.575,A -85,B 0,C 180,E1 9152.651,E2 9152.651} C_VEL
LIN {X 0,Y 241.655,Z 871.909,A -85,B 0,C 180,E1 9150.809,E2 9150.809} C_VEL
LIN {X 0,Y 232.556,Z 889.114,A -85,B 0,C 180,E1 9148.585,E2 9148.585} C_VEL
LIN {X 0,Y 223.128,Z 904.71,A -85,B 0,C 180,E1 9145.994,E2 9145.994} C_VEL
LIN {X 0,Y 213.179,Z 919.379,A -85,B 0,C 180,E1 9142.874,E2 9142.874} C_VEL
LIN {X 0,Y 203.272,Z 932.601,A -85,B 0,C 180,E1 9139.242,E2 9139.242} C_VEL
LIN {X 0,Y 193.458,Z 944.653,A -85,B 0,C 180,E1 9134.922,E2 9134.922} C_VEL
LIN {X 0,Y 184.637,Z 954.854,A -85,B 0,C 180,E1 9130.12,E2 9130.12} C_VEL
LIN {X 0,Y 176.181,Z 964.228,A -85,B 0,C 180,E1 9124.181,E2 9124.181} C_VEL
LIN {X 0,Y 169.533,Z 971.555,A -85,B 0,C 180,E1 9117.768,E2 9117.768} C_VEL
LIN {X 0,Y 164.669,Z 977.182,A -85,B 0,C 180,E1 9110.758,E2 9110.758} C_VEL
LIN {X 0,Y 161.792,Z 980.972,A -85,B 0,C 180,E1 9103.58,E2 9103.58} C_VEL
LIN {X 0,Y 160.55,Z 983.103,A -85,B 0,C 180,E1 9096.434,E2 9096.434} C_VEL
LIN {X 0,Y 160.322,Z 983.775,A -85,B 0,C 180,E1 9089.998,E2 9089.998} C_VEL
LIN {X 0,Y 160.544,Z 983.132,A -85,B 0,C 180,E1 9083.562,E2 9083.562} C_VEL
LIN {X 0,Y 161.77,Z 981.039,A -85,B 0,C 180,E1 9076.414,E2 9076.414} C_VEL
LIN {X 0,Y 164.583,Z 977.346,A -85,B 0,C 180,E1 9069.322,E2 9069.322} C_VEL
LIN {X 0,Y 169.476,Z 971.692,A -85,B 0,C 180,E1 9062.218,E2 9062.218} C_VEL
LIN {X 0,Y 176.107,Z 964.388,A -85,B 0,C 180,E1 9055.798,E2 9055.798} C_VEL
LIN {X 0,Y 184.084,Z 955.557,A -85,B 0,C 180,E1 9050.137,E2 9050.137} C_VEL
LIN {X 0,Y 193.05,Z 945.266,A -85,B 0,C 180,E1 9045.2,E2 9045.2} C_VEL
LIN {X 0,Y 202.576,Z 933.651,A -85,B 0,C 180,E1 9040.958,E2 9040.958} C_VEL
LIN {X 0,Y 212.435,Z 920.642,A -85,B 0,C 180,E1 9037.302,E2 9037.302} C_VEL
LIN {X 0,Y 222.342,Z 906.222,A -85,B 0,C 180,E1 9034.161,E2 9034.161} C_VEL
LIN {X 0,Y 228.34,Z 896.402,A -85,B 0,C 180,E1 9032.382,E2 9032.382} C_VEL
LIN {X 0,Y 222.463,Z 899.604,A -85,B 0,C 180,E1 9031.123,E2 9031.123} C_VEL
LIN {X 0,Y 213.207,Z 904.339,A -85,B 0,C 180,E1 9028.884,E2 9028.884} C_VEL
LIN {X 0,Y 208.227,Z 906.78,A -85,B 0,C 180,E1 9027.45,E2 9027.45} C_VEL
LIN {X 0,Y 200.827,Z 910.328,A -85,B 0,C 180,E1 9025.037,E2 9025.037} C_VEL
LIN {X 0,Y 196.481,Z 912.306,A -85,B 0,C 180,E1 9023.387,E2 9023.387} C_VEL
LIN {X 0,Y 190.04,Z 915.25,A -85,B 0,C 180,E1 9020.521,E2 9020.521} C_VEL
LIN {X 0,Y 182.414,Z 918.884,A -85,B 0,C 180,E1 9016.234,E2 9016.234} C_VEL
LIN {X 0,Y 179.89,Z 920.086,A -85,B 0,C 180,E1 9014.485,E2 9014.485} C_VEL
LIN {X 0,Y 175.813,Z 922.183,A -85,B 0,C 180,E1 9011.149,E2 9011.149} C_VEL
LIN {X 0,Y 174.508,Z 922.882,A -85,B 0,C 180,E1 9009.777,E2 9009.777} C_VEL
LIN {X 0,Y 170.846,Z 925.591,A -85,B 0,C 180,E1 9007.216,E2 9007.216} C_VEL
LIN {X 0,Y 163.825,Z 931.446,A -85,B 0,C 180,E1 9002.405,E2 9002.405} C_VEL
LIN {X 0,Y 162.017,Z 933.182,A -85,B 0,C 180,E1 8999.855,E2 8999.855} C_VEL
LIN {X 0,Y 161.844,Z 933.45,A -85,B 0,C 180,E1 8999.089,E2 8999.089} C_VEL
LIN {X 0,Y 160.984,Z 936.405,A -85,B 0,C 180,E1 8992.147,E2 8992.147} C_VEL
LIN {X 0,Y 161.743,Z 937.689,A -85,B 0,C 180,E1 8988.591,E2 8988.591} C_VEL
LIN {X 0,Y 165.33,Z 940.281,A -85,B 0,C 180,E1 8981.306,E2 8981.306} C_VEL
LIN {X 0,Y 178.178,Z 943.331,A -85,B 0,C 180,E1 8970.409,E2 8970.409} C_VEL
LIN {X 0,Y 191.995,Z 944.372,A -85,B 0,C 180,E1 8963.952,E2 8963.952} C_VEL
LIN {X 0,Y 195.717,Z 944.519,A -85,B 0,C 180,E1 8962.577,E2 8962.577} C_VEL
LIN {X 0,Y 185.735,Z 956.628,A -85,B 0,C 180,E1 8958.443,E2 8958.443} C_VEL
LIN {X 0,Y 175.576,Z 968.277,A -85,B 0,C 180,E1 8953.11,E2 8953.11} C_VEL
LIN {X 0,Y 166.668,Z 978.238,A -85,B 0,C 180,E1 8946.866,E2 8946.866} C_VEL
LIN {X 0,Y 159.858,Z 986.119,A -85,B 0,C 180,E1 8940.027,E2 8940.027} C_VEL
LIN {X 0,Y 155.26,Z 992.128,A -85,B 0,C 180,E1 8932.732,E2 8932.732} C_VEL
LIN {X 0,Y 152.829,Z 996.389,A -85,B 0,C 180,E1 8925.173,E2 8925.173} C_VEL
LIN {X 0,Y 152.255,Z 998.901,A -85,B 0,C 180,E1 8917.929,E2 8917.929} C_VEL
LIN {X 0,Y 152.442,Z 999.751,A -85,B 0,C 180,E1 8912.257,E2 8912.257} C_VEL
LIN {X 0,Y 152.441,Z 999.747,A -85,B 0,C 180,E1 8907.747,E2 8907.747} C_VEL
LIN {X 0,Y 152.236,Z 998.813,A -85,B 0,C 180,E1 8901.694,E2 8901.694} C_VEL
LIN {X 0,Y 152.871,Z 996.191,A -85,B 0,C 180,E1 8894.447,E2 8894.447} C_VEL
LIN {X 0,Y 155.399,Z 991.821,A -85,B 0,C 180,E1 8886.893,E2 8886.893} C_VEL
LIN {X 0,Y 160.113,Z 985.697,A -85,B 0,C 180,E1 8879.616,E2 8879.616} C_VEL
LIN {X 0,Y 166.627,Z 978.16,A -85,B 0,C 180,E1 8873.128,E2 8873.128} C_VEL
LIN {X 0,Y 175.528,Z 968.178,A -85,B 0,C 180,E1 8866.88,E2 8866.88} C_VEL
LIN {X 0,Y 185.687,Z 956.511,A -85,B 0,C 180,E1 8861.545,E2 8861.545} C_VEL
LIN {X 0,Y 196.018,Z 943.947,A -85,B 0,C 180,E1 8857.278,E2 8857.278} C_VEL
LIN {X 0,Y 206.636,Z 929.958,A -85,B 0,C 180,E1 8853.671,E2 8853.671} C_VEL
LIN {X 0,Y 217.321,Z 914.483,A -85,B 0,C 180,E1 8850.646,E2 8850.646} C_VEL
LIN {X 0,Y 227.819,Z 897.356,A -85,B 0,C 180,E1 8848.1,E2 8848.1} C_VEL
LIN {X 0,Y 237.178,Z 879.855,A -85,B 0,C 180,E1 8846.115,E2 8846.115} C_VEL
LIN {X 0,Y 245.516,Z 861.732,A -85,B 0,C 180,E1 8844.544,E2 8844.544} C_VEL
LIN {X 0,Y 252.955,Z 842.454,A -85,B 0,C 180,E1 8843.283,E2 8843.283} C_VEL
LIN {X 0,Y 259.345,Z 821.728,A -85,B 0,C 180,E1 8842.293,E2 8842.293} C_VEL
LIN {X 0,Y 264.231,Z 800.339,A -85,B 0,C 180,E1 8841.562,E2 8841.562} C_VEL
LIN {X 0,Y 267.26,Z 780.318,A -85,B 0,C 180,E1 8841.085,E2 8841.085} C_VEL
LIN {X 0,Y 270.637,Z 751.579,A -85,B 0,C 180,E1 8840.806,E2 8840.806} C_VEL
LIN {X 0,Y 268.797,Z 724.453,A -85,B 0,C 180,E1 8837.577,E2 8837.577} C_VEL
LIN {X 0,Y 268.331,Z 697.529,A -85,B 0,C 180,E1 8834.746,E2 8834.746} C_VEL
LIN {X 0,Y 269.053,Z 667.229,A -85,B 0,C 180,E1 8832.02,E2 8832.02} C_VEL
LIN {X 0,Y 269.074,Z 665.663,A -85,B 0,C 180,E1 8831.847,E2 8831.847} C_VEL
LIN {X 0,Y 266.951,Z 649.353,A -85,B 0,C 180,E1 8826.505,E2 8826.505} C_VEL
LIN {X 0,Y 266.913,Z 634.807,A -85,B 0,C 180,E1 8820.644,E2 8820.644} C_VEL
LIN {X 0,Y 268.449,Z 625.846,A -85,B 0,C 180,E1 8816.369,E2 8816.369} C_VEL
LIN {X 0,Y 270.574,Z 619.792,A -85,B 0,C 180,E1 8813.049,E2 8813.049} C_VEL
LIN {X 0,Y 272.167,Z 622.685,A -85,B 0,C 180,E1 8810.164,E2 8810.164} C_VEL
LIN {X 0,Y 274.313,Z 627.09,A -85,B 0,C 180,E1 8807.26,E2 8807.26} C_VEL
LIN {X 0,Y 277.186,Z 632.913,A -85,B 0,C 180,E1 8804.25,E2 8804.25} C_VEL
LIN {X 0,Y 280.814,Z 640.807,A -85,B 0,C 180,E1 8801.141,E2 8801.141} C_VEL
LIN {X 0,Y 267.653,Z 775.956,A -85,B 0,C 180,E1 8798.378,E2 8798.378} C_VEL
LIN {X 0,Y 264.223,Z 796.283,A -85,B 0,C 180,E1 8797.739,E2 8797.739} C_VEL
LIN {X 0,Y 259.349,Z 816.546,A -85,B 0,C 180,E1 8796.844,E2 8796.844} C_VEL
LIN {X 0,Y 253.381,Z 835.615,A -85,B 0,C 180,E1 8795.716,E2 8795.716} C_VEL
LIN {X 0,Y 246.313,Z 853.974,A -85,B 0,C 180,E1 8794.309,E2 8794.309} C_VEL
LIN {X 0,Y 237.839,Z 872.313,A -85,B 0,C 180,E1 8792.5,E2 8792.5} C_VEL
LIN {X 0,Y 228.463,Z 889.521,A -85,B 0,C 180,E1 8790.308,E2 8790.308} C_VEL
LIN {X 0,Y 218.718,Z 905.12,A -85,B 0,C 180,E1 8787.746,E2 8787.746} C_VEL
LIN {X 0,Y 208.398,Z 919.792,A -85,B 0,C 180,E1 8784.647,E2 8784.647} C_VEL
LIN {X 0,Y 198.081,Z 933.016,A -85,B 0,C 180,E1 8781.016,E2 8781.016} C_VEL
LIN {X 0,Y 188.007,Z 944.843,A -85,B 0,C 180,E1 8776.766,E2 8776.766} C_VEL
LIN {X 0,Y 178.505,Z 955.271,A -85,B 0,C 180,E1 8771.799,E2 8771.799} C_VEL
LIN {X 0,Y 169.523,Z 964.646,A -85,B 0,C 180,E1 8765.724,E2 8765.724} C_VEL
LIN {X 0,Y 162.092,Z 972.305,A -85,B 0,C 180,E1 8758.758,E2 8758.758} C_VEL
LIN {X 0,Y 156.852,Z 977.934,A -85,B 0,C 180,E1 8751.304,E2 8751.304} C_VEL
LIN {X 0,Y 153.864,Z 981.539,A -85,B 0,C 180,E1 8743.91,E2 8743.91} C_VEL
LIN {X 0,Y 152.589,Z 983.516,A -85,B 0,C 180,E1 8736.772,E2 8736.772} C_VEL
LIN {X 0,Y 152.332,Z 984.187,A -85,B 0,C 180,E1 8729.998,E2 8729.998} C_VEL
LIN {X 0,Y 152.582,Z 983.544,A -85,B 0,C 180,E1 8723.224,E2 8723.224} C_VEL
LIN {X 0,Y 153.947,Z 981.453,A -85,B 0,C 180,E1 8715.71,E2 8715.71} C_VEL
LIN {X 0,Y 157.012,Z 977.791,A -85,B 0,C 180,E1 8708.323,E2 8708.323} C_VEL
LIN {X 0,Y 162.339,Z 972.108,A -85,B 0,C 180,E1 8700.883,E2 8700.883} C_VEL
LIN {X 0,Y 169.449,Z 964.803,A -85,B 0,C 180,E1 8694.254,E2 8694.254} C_VEL
LIN {X 0,Y 177.925,Z 955.971,A -85,B 0,C 180,E1 8688.46,E2 8688.46} C_VEL
LIN {X 0,Y 187.353,Z 945.706,A -85,B 0,C 180,E1 8683.462,E2 8683.462} C_VEL
LIN {X 0,Y 197.362,Z 934.061,A -85,B 0,C 180,E1 8679.182,E2 8679.182} C_VEL
LIN {X 0,Y 207.633,Z 921.049,A -85,B 0,C 180,E1 8675.527,E2 8675.527} C_VEL
LIN {X 0,Y 217.912,Z 906.625,A -85,B 0,C 180,E1 8672.405,E2 8672.405} C_VEL
LIN {X 0,Y 218.42,Z 905.775,A -85,B 0,C 180,E1 8672.229,E2 8672.229} C_VEL
LIN {X 0,Y 209.502,Z 909.987,A -85,B 0,C 180,E1 8670.074,E2 8670.074} C_VEL
LIN {X 0,Y 197.979,Z 915.262,A -85,B 0,C 180,E1 8666.711,E2 8666.711} C_VEL
LIN {X 0,Y 192.187,Z 917.795,A -85,B 0,C 180,E1 8664.596,E2 8664.596} C_VEL
LIN {X 0,Y 185.193,Z 920.687,A -85,B 0,C 180,E1 8661.539,E2 8661.539} C_VEL
LIN {X 0,Y 177.907,Z 923.915,A -85,B 0,C 180,E1 8657.668,E2 8657.668} C_VEL
LIN {X 0,Y 174.844,Z 925.284,A -85,B 0,C 180,E1 8655.592,E2 8655.592} C_VEL
LIN {X 0,Y 170.255,Z 927.522,A -85,B 0,C 180,E1 8651.862,E2 8651.862} C_VEL
LIN {X 0,Y 165.428,Z 930.253,A -85,B 0,C 180,E1 8646.595,E2 8646.595} C_VEL
LIN {X 0,Y 164.158,Z 931.137,A -85,B 0,C 180,E1 8644.542,E2 8644.542} C_VEL
LIN {X 0,Y 161.982,Z 933.187,A -85,B 0,C 180,E1 8639.997,E2 8639.997} C_VEL
LIN {X 0,Y 161.844,Z 933.45,A -85,B 0,C 180,E1 8639.089,E2 8639.089} C_VEL
LIN {X 0,Y 161.009,Z 934.482,A -85,B 0,C 180,E1 8637.566,E2 8637.566} C_VEL
LIN {X 0,Y 157.351,Z 938.254,A -85,B 0,C 180,E1 8634.837,E2 8634.837} C_VEL
LIN {X 0,Y 155.061,Z 940.774,A -85,B 0,C 180,E1 8632.658,E2 8632.658} C_VEL
LIN {X 0,Y 154.811,Z 941.522,A -85,B 0,C 180,E1 8631.308,E2 8631.308} C_VEL
LIN {X 0,Y 158.499,Z 944.879,A -85,B 0,C 180,E1 8621.615,E2 8621.615} C_VEL
LIN {X 0,Y 171.688,Z 948.065,A -85,B 0,C 180,E1 8609.945,E2 8609.945} C_VEL
LIN {X 0,Y 185.63,Z 949.192,A -85,B 0,C 180,E1 8603.283,E2 8603.283} C_VEL
LIN {X 0,Y 186.469,Z 949.314,A -85,B 0,C 180,E1 8602.905,E2 8602.905} C_VEL
LIN {X 0,Y 175.104,Z 962.015,A -85,B 0,C 180,E1 8597.931,E2 8597.931} C_VEL
LIN {X 0,Y 165.135,Z 972.592,A -85,B 0,C 180,E1 8592.23,E2 8592.23} C_VEL
LIN {X 0,Y 156.935,Z 981.169,A -85,B 0,C 180,E1 8585.886,E2 8585.886} C_VEL
LIN {X 0,Y 150.454,Z 988.296,A -85,B 0,C 180,E1 8578.589,E2 8578.589} C_VEL
LIN {X 0,Y 146.196,Z 993.833,A -85,B 0,C 180,E1 8570.416,E2 8570.416} C_VEL
LIN {X 0,Y 144.434,Z 997.349,A -85,B 0,C 180,E1 8562.394,E2 8562.394} C_VEL
LIN {X 0,Y 144.318,Z 999.007,A -85,B 0,C 180,E1 8555.568,E2 8555.568} C_VEL
LIN {X 0,Y 144.504,Z 999.457,A -85,B 0,C 180,E1 8549.606,E2 8549.606} C_VEL
LIN {X 0,Y 144.272,Z 998.846,A -85,B 0,C 180,E1 8543.636,E2 8543.636} C_VEL
LIN {X 0,Y 144.546,Z 996.951,A -85,B 0,C 180,E1 8536.4,E2 8536.4} C_VEL
LIN {X 0,Y 146.623,Z 993.145,A -85,B 0,C 180,E1 8528.395,E2 8528.395} C_VEL
LIN {X 0,Y 150.969,Z 987.617,A -85,B 0,C 180,E1 8520.655,E2 8520.655} C_VEL
LIN {X 0,Y 157.66,Z 980.265,A -85,B 0,C 180,E1 8513.409,E2 8513.409} C_VEL
LIN {X 0,Y 166.55,Z 970.92,A -85,B 0,C 180,E1 8506.816,E2 8506.816} C_VEL
LIN {X 0,Y 176.197,Z 960.609,A -85,B 0,C 180,E1 8501.494,E2 8501.494} C_VEL
LIN {X 0,Y 186.578,Z 948.985,A -85,B 0,C 180,E1 8497.017,E2 8497.017} C_VEL
LIN {X 0,Y 197.979,Z 935.113,A -85,B 0,C 180,E1 8493.036,E2 8493.036} C_VEL
LIN {X 0,Y 209.187,Z 920.04,A -85,B 0,C 180,E1 8489.807,E2 8489.807} C_VEL
LIN {X 0,Y 219.795,Z 904.051,A -85,B 0,C 180,E1 8487.213,E2 8487.213} C_VEL
LIN {X 0,Y 229.681,Z 887.114,A -85,B 0,C 180,E1 8485.115,E2 8485.115} C_VEL
LIN {X 0,Y 239.056,Z 868.459,A -85,B 0,C 180,E1 8483.358,E2 8483.358} C_VEL
LIN {X 0,Y 247.002,Z 849.727,A -85,B 0,C 180,E1 8482.033,E2 8482.033} C_VEL
LIN {X 0,Y 253.753,Z 830.362,A -85,B 0,C 180,E1 8481.012,E2 8481.012} C_VEL
LIN {X 0,Y 259.377,Z 809.571,A -85,B 0,C 180,E1 8480.217,E2 8480.217} C_VEL
LIN {X 0,Y 263.453,Z 787.808,A -85,B 0,C 180,E1 8479.605,E2 8479.605} C_VEL
LIN {X 0,Y 266.612,Z 762.211,A -85,B 0,C 180,E1 8479.288,E2 8479.288} C_VEL
LIN {X 0,Y 267.599,Z 753.633,A -85,B 0,C 180,E1 8479.21,E2 8479.21} C_VEL
LIN {X 0,Y 266.258,Z 727.168,A -85,B 0,C 180,E1 8476.05,E2 8476.05} C_VEL
LIN {X 0,Y 266.149,Z 700.604,A -85,B 0,C 180,E1 8473.234,E2 8473.234} C_VEL
LIN {X 0,Y 267.134,Z 670.691,A -85,B 0,C 180,E1 8470.459,E2 8470.459} C_VEL
LIN {X 0,Y 265.65,Z 655.969,A -85,B 0,C 180,E1 8465.561,E2 8465.561} C_VEL
LIN {X 0,Y 266.004,Z 641.956,A -85,B 0,C 180,E1 8459.892,E2 8459.892} C_VEL
LIN {X 0,Y 267.741,Z 633.209,A -85,B 0,C 180,E1 8455.716,E2 8455.716} C_VEL
LIN {X 0,Y 269.654,Z 628.067,A -85,B 0,C 180,E1 8452.864,E2 8452.864} C_VEL
LIN {X 0,Y 270.97,Z 630.54,A -85,B 0,C 180,E1 8450.442,E2 8450.442} C_VEL
LIN {X 0,Y 273.045,Z 634.994,A -85,B 0,C 180,E1 8447.522,E2 8447.522} C_VEL
LIN {X 0,Y 276.041,Z 641.464,A -85,B 0,C 180,E1 8444.29,E2 8444.29} C_VEL
LIN {X 0,Y 277.859,Z 645.839,A -85,B 0,C 180,E1 8442.608,E2 8442.608} C_VEL
LIN {X 0,Y 264.799,Z 776.384,A -85,B 0,C 180,E1 8439.983,E2 8439.983} C_VEL
LIN {X 0,Y 261.298,Z 796.648,A -85,B 0,C 180,E1 8439.362,E2 8439.362} C_VEL
LIN {X 0,Y 256.294,Z 816.978,A -85,B 0,C 180,E1 8438.486,E2 8438.486} C_VEL
LIN {X 0,Y 249.787,Z 837.113,A -85,B 0,C 180,E1 8437.314,E2 8437.314} C_VEL
LIN {X 0,Y 242.271,Z 855.85,A -85,B 0,C 180,E1 8435.884,E2 8435.884} C_VEL
LIN {X 0,Y 234.237,Z 872.716,A -85,B 0,C 180,E1 8434.243,E2 8434.243} C_VEL
LIN {X 0,Y 224.586,Z 889.928,A -85,B 0,C 180,E1 8432.092,E2 8432.092} C_VEL
LIN {X 0,Y 214.522,Z 905.53,A -85,B 0,C 180,E1 8429.569,E2 8429.569} C_VEL
LIN {X 0,Y 203.828,Z 920.205,A -85,B 0,C 180,E1 8426.501,E2 8426.501} C_VEL
LIN {X 0,Y 193.089,Z 933.431,A -85,B 0,C 180,E1 8422.884,E2 8422.884} C_VEL
LIN {X 0,Y 182.547,Z 945.26,A -85,B 0,C 180,E1 8418.621,E2 8418.621} C_VEL
LIN {X 0,Y 172.466,Z 955.757,A -85,B 0,C 180,E1 8413.557,E2 8413.557} C_VEL
LIN {X 0,Y 162.999,Z 965.065,A -85,B 0,C 180,E1 8407.391,E2 8407.391} C_VEL
LIN {X 0,Y 155.027,Z 972.723,A -85,B 0,C 180,E1 8400.201,E2 8400.201} C_VEL
LIN {X 0,Y 149.34,Z 978.352,A -85,B 0,C 180,E1 8392.432,E2 8392.432} C_VEL
LIN {X 0,Y 146.055,Z 981.954,A -85,B 0,C 180,E1 8384.67,E2 8384.67} C_VEL
LIN {X 0,Y 144.634,Z 983.929,A -85,B 0,C 180,E1 8377.146,E2 8377.146} C_VEL
LIN {X 0,Y 144.337,Z 984.579,A -85,B 0,C 180,E1 8370.395,E2 8370.395} C_VEL
LIN {X 0,Y 144.588,Z 984.02,A -85,B 0,C 180,E1 8363.247,E2 8363.247} C_VEL
LIN {X 0,Y 145.921,Z 982.17,A -85,B 0,C 180,E1 8355.717,E2 8355.717} C_VEL
LIN {X 0,Y 149.087,Z 978.666,A -85,B 0,C 180,E1 8347.939,E2 8347.939} C_VEL
LIN {X 0,Y 154.324,Z 973.423,A -85,B 0,C 180,E1 8340.499,E2 8340.499} C_VEL
LIN {X 0,Y 161.234,Z 966.784,A -85,B 0,C 180,E1 8333.903,E2 8333.903} C_VEL
LIN {X 0,Y 170.397,Z 957.884,A -85,B 0,C 180,E1 8327.559,E2 8327.559} C_VEL
LIN {X 0,Y 180.701,Z 947.356,A -85,B 0,C 180,E1 8322.142,E2 8322.142} C_VEL
LIN {X 0,Y 191.322,Z 935.67,A -85,B 0,C 180,E1 8317.695,E2 8317.695} C_VEL
LIN {X 0,Y 201.925,Z 922.928,A -85,B 0,C 180,E1 8314.024,E2 8314.024} C_VEL
LIN {X 0,Y 208.395,Z 914.369,A -85,B 0,C 180,E1 8312.033,E2 8312.033} C_VEL
LIN {X 0,Y 194.508,Z 920.287,A -85,B 0,C 180,E1 8308.225,E2 8308.225} C_VEL
LIN {X 0,Y 181.679,Z 925.492,A -85,B 0,C 180,E1 8303.344,E2 8303.344} C_VEL
LIN {X 0,Y 172.502,Z 929.135,A -85,B 0,C 180,E1 8298.59,E2 8298.59} C_VEL
LIN {X 0,Y 165.145,Z 932.333,A -85,B 0,C 180,E1 8293.302,E2 8293.302} C_VEL
LIN {X 0,Y 162.306,Z 933.748,A -85,B 0,C 180,E1 8290.651,E2 8290.651} C_VEL
LIN {X 0,Y 159.111,Z 935.542,A -85,B 0,C 180,E1 8286.495,E2 8286.495} C_VEL
LIN {X 0,Y 155.896,Z 938.053,A -85,B 0,C 180,E1 8280.736,E2 8280.736} C_VEL
LIN {X 0,Y 155.237,Z 938.964,A -85,B 0,C 180,E1 8278.155,E2 8278.155} C_VEL
LIN {X 0,Y 154.635,Z 941.27,A -85,B 0,C 180,E1 8272.197,E2 8272.197} C_VEL
LIN {X 0,Y 154.811,Z 941.522,A -85,B 0,C 180,E1 8271.308,E2 8271.308} C_VEL
LIN {X 0,Y 154.551,Z 942.501,A -85,B 0,C 180,E1 8269.687,E2 8269.687} C_VEL
LIN {X 0,Y 151.841,Z 946.254,A -85,B 0,C 180,E1 8266.39,E2 8266.39} C_VEL
LIN {X 0,Y 150.665,Z 948.459,A -85,B 0,C 180,E1 8263.988,E2 8263.988} C_VEL
LIN {X 0,Y 150.955,Z 948.986,A -85,B 0,C 180,E1 8262.875,E2 8262.875} C_VEL
LIN {X 0,Y 165.044,Z 952.516,A -85,B 0,C 180,E1 8249.411,E2 8249.411} C_VEL
LIN {X 0,Y 177.184,Z 953.698,A -85,B 0,C 180,E1 8243.259,E2 8243.259} C_VEL
LIN {X 0,Y 166.178,Z 965.109,A -85,B 0,C 180,E1 8238.255,E2 8238.255} C_VEL
LIN {X 0,Y 156.141,Z 975.047,A -85,B 0,C 180,E1 8232.253,E2 8232.253} C_VEL
LIN {X 0,Y 147.605,Z 983.451,A -85,B 0,C 180,E1 8225.157,E2 8225.157} C_VEL
LIN {X 0,Y 141.397,Z 989.955,A -85,B 0,C 180,E1 8217.366,E2 8217.366} C_VEL
LIN {X 0,Y 137.683,Z 994.698,A -85,B 0,C 180,E1 8209.077,E2 8209.077} C_VEL
LIN {X 0,Y 136.326,Z 997.543,A -85,B 0,C 180,E1 8200.995,E2 8200.995} C_VEL
LIN {X 0,Y 136.395,Z 998.847,A -85,B 0,C 180,E1 8193.785,E2 8193.785} C_VEL
LIN {X 0,Y 136.48,Z 998.973,A -85,B 0,C 180,E1 8188.323,E2 8188.323} C_VEL
LIN {X 0,Y 136.25,Z 998.207,A -85,B 0,C 180,E1 8181.987,E2 8181.987} C_VEL
LIN {X 0,Y 136.934,Z 995.858,A -85,B 0,C 180,E1 8173.893,E2 8173.893} C_VEL
LIN {X 0,Y 139.796,Z 991.77,A -85,B 0,C 180,E1 8165.494,E2 8165.494} C_VEL
LIN {X 0,Y 145.123,Z 985.931,A -85,B 0,C 180,E1 8157.496,E2 8157.496} C_VEL
LIN {X 0,Y 152.852,Z 978.174,A -85,B 0,C 180,E1 8150.132,E2 8150.132} C_VEL
LIN {X 0,Y 162.235,Z 968.919,A -85,B 0,C 180,E1 8143.86,E2 8143.86} C_VEL
LIN {X 0,Y 172.695,Z 958.25,A -85,B 0,C 180,E1 8138.594,E2 8138.594} C_VEL
LIN {X 0,Y 184.463,Z 945.446,A -85,B 0,C 180,E1 8133.974,E2 8133.974} C_VEL
LIN {X 0,Y 195.816,Z 931.925,A -85,B 0,C 180,E1 8130.356,E2 8130.356} C_VEL
LIN {X 0,Y 207.146,Z 917.002,A -85,B 0,C 180,E1 8127.363,E2 8127.363} C_VEL
LIN {X 0,Y 218.207,Z 900.549,A -85,B 0,C 180,E1 8124.873,E2 8124.873} C_VEL
LIN {X 0,Y 228.428,Z 883.03,A -85,B 0,C 180,E1 8122.874,E2 8122.874} C_VEL
LIN {X 0,Y 237.241,Z 865.363,A -85,B 0,C 180,E1 8121.348,E2 8121.348} C_VEL
LIN {X 0,Y 244.955,Z 847.087,A -85,B 0,C 180,E1 8120.15,E2 8120.15} C_VEL
LIN {X 0,Y 251.926,Z 826.815,A -85,B 0,C 180,E1 8119.167,E2 8119.167} C_VEL
LIN {X 0,Y 257.307,Z 806.413,A -85,B 0,C 180,E1 8118.452,E2 8118.452} C_VEL
LIN {X 0,Y 261.103,Z 785.774,A -85,B 0,C 180,E1 8117.914,E2 8117.914} C_VEL
LIN {X 0,Y 264.531,Z 758.214,A -85,B 0,C 180,E1 8117.635,E2 8117.635} C_VEL
LIN {X 0,Y 264.774,Z 755.572,A -85,B 0,C 180,E1 8117.569,E2 8117.569} C_VEL
LIN {X 0,Y 263.913,Z 730.007,A -85,B 0,C 180,E1 8114.508,E2 8114.508} C_VEL
LIN {X 0,Y 264.155,Z 703.68,A -85,B 0,C 180,E1 8111.697,E2 8111.697} C_VEL
LIN {X 0,Y 265.374,Z 675.877,A -85,B 0,C 180,E1 8109.105,E2 8109.105} C_VEL
LIN {X 0,Y 264.426,Z 662.717,A -85,B 0,C 180,E1 8104.663,E2 8104.663} C_VEL
LIN {X 0,Y 265.141,Z 649.103,A -85,B 0,C 180,E1 8099.135,E2 8099.135} C_VEL
LIN {X 0,Y 267.132,Z 640.383,A -85,B 0,C 180,E1 8094.953,E2 8094.953} C_VEL
LIN {X 0,Y 268.715,Z 636.265,A -85,B 0,C 180,E1 8092.732,E2 8092.732} C_VEL
LIN {X 0,Y 269.78,Z 638.391,A -85,B 0,C 180,E1 8090.722,E2 8090.722} C_VEL
LIN {X 0,Y 271.702,Z 642.717,A -85,B 0,C 180,E1 8087.891,E2 8087.891} C_VEL
LIN {X 0,Y 274.691,Z 649.519,A -85,B 0,C 180,E1 8084.536,E2 8084.536} C_VEL
LIN {X 0,Y 275.086,Z 650.895,A -85,B 0,C 180,E1 8084.105,E2 8084.105} C_VEL
LIN {X 0,Y 262.144,Z 776.918,A -85,B 0,C 180,E1 8081.621,E2 8081.621} C_VEL
LIN {X 0,Y 258.559,Z 797.152,A -85,B 0,C 180,E1 8081.015,E2 8081.015} C_VEL
LIN {X 0,Y 253.454,Z 817.407,A -85,B 0,C 180,E1 8080.168,E2 8080.168} C_VEL
LIN {X 0,Y 246.808,Z 837.505,A -85,B 0,C 180,E1 8079.03,E2 8079.03} C_VEL
LIN {X 0,Y 239.341,Z 855.743,A -85,B 0,C 180,E1 8077.683,E2 8077.683} C_VEL
LIN {X 0,Y 230.858,Z 873.12,A -85,B 0,C 180,E1 8076.04,E2 8076.04} C_VEL
LIN {X 0,Y 221.165,Z 889.946,A -85,B 0,C 180,E1 8073.99,E2 8073.99} C_VEL
LIN {X 0,Y 210.976,Z 905.33,A -85,B 0,C 180,E1 8071.569,E2 8071.569} C_VEL
LIN {X 0,Y 200.202,Z 919.712,A -85,B 0,C 180,E1 8068.648,E2 8068.648} C_VEL
LIN {X 0,Y 188.989,Z 933.093,A -85,B 0,C 180,E1 8065.086,E2 8065.086} C_VEL
LIN {X 0,Y 177.916,Z 945.057,A -85,B 0,C 180,E1 8060.851,E2 8060.851} C_VEL
LIN {X 0,Y 167.304,Z 955.595,A -85,B 0,C 180,E1 8055.818,E2 8055.818} C_VEL
LIN {X 0,Y 157.084,Z 965.059,A -85,B 0,C 180,E1 8049.53,E2 8049.53} C_VEL
LIN {X 0,Y 148.782,Z 972.469,A -85,B 0,C 180,E1 8042.52,E2 8042.52} C_VEL
LIN {X 0,Y 142.619,Z 978.039,A -85,B 0,C 180,E1 8034.873,E2 8034.873} C_VEL
LIN {X 0,Y 138.674,Z 981.916,A -85,B 0,C 180,E1 8026.76,E2 8026.76} C_VEL
LIN {X 0,Y 136.785,Z 984.216,A -85,B 0,C 180,E1 8018.404,E2 8018.404} C_VEL
LIN {X 0,Y 136.348,Z 984.947,A -85,B 0,C 180,E1 8011.258,E2 8011.258} C_VEL
LIN {X 0,Y 136.528,Z 984.624,A -85,B 0,C 180,E1 8004.113,E2 8004.113} C_VEL
LIN {X 0,Y 137.685,Z 983.09,A -85,B 0,C 180,E1 7996.56,E2 7996.56} C_VEL
LIN {X 0,Y 140.736,Z 979.868,A -85,B 0,C 180,E1 7988.317,E2 7988.317} C_VEL
LIN {X 0,Y 146.315,Z 974.713,A -85,B 0,C 180,E1 7980.073,E2 7980.073} C_VEL
LIN {X 0,Y 153.873,Z 967.982,A -85,B 0,C 180,E1 7972.818,E2 7972.818} C_VEL
LIN {X 0,Y 162.917,Z 959.797,A -85,B 0,C 180,E1 7966.575,E2 7966.575} C_VEL
LIN {X 0,Y 173.261,Z 949.934,A -85,B 0,C 180,E1 7961.139,E2 7961.139} C_VEL
LIN {X 0,Y 184.885,Z 937.88,A -85,B 0,C 180,E1 7956.31,E2 7956.31} C_VEL
LIN {X 0,Y 196.536,Z 924.517,A -85,B 0,C 180,E1 7952.378,E2 7952.378} C_VEL
LIN {X 0,Y 198.243,Z 922.331,A -85,B 0,C 180,E1 7951.807,E2 7951.807} C_VEL
LIN {X 0,Y 189.009,Z 925.914,A -85,B 0,C 180,E1 7949.123,E2 7949.123} C_VEL
LIN {X 0,Y 177.526,Z 930.247,A -85,B 0,C 180,E1 7944.932,E2 7944.932} C_VEL
LIN {X 0,Y 167.489,Z 934.036,A -85,B 0,C 180,E1 7939.894,E2 7939.894} C_VEL
LIN {X 0,Y 159.325,Z 937.255,A -85,B 0,C 180,E1 7934.168,E2 7934.168} C_VEL
LIN {X 0,Y 153.356,Z 940.132,A -85,B 0,C 180,E1 7927.87,E2 7927.87} C_VEL
LIN {X 0,Y 149.489,Z 942.959,A -85,B 0,C 180,E1 7920.767,E2 7920.767} C_VEL
LIN {X 0,Y 148.225,Z 946.075,A -85,B 0,C 180,E1 7911.857,E2 7911.857} C_VEL
LIN {X 0,Y 150.955,Z 948.986,A -85,B 0,C 180,E1 7902.875,E2 7902.875} C_VEL
LIN {X 0,Y 152.025,Z 950.364,A -85,B 0,C 180,E1 7900.003,E2 7900.003} C_VEL
LIN {X 0,Y 153.809,Z 955.401,A -85,B 0,C 180,E1 7892.728,E2 7892.728} C_VEL
LIN {X 0,Y 156.426,Z 956.493,A -85,B 0,C 180,E1 7890.072,E2 7890.072} C_VEL
LIN {X 0,Y 167.824,Z 957.865,A -85,B 0,C 180,E1 7883.626,E2 7883.626} C_VEL
LIN {X 0,Y 156.68,Z 968.597,A -85,B 0,C 180,E1 7878.303,E2 7878.303} C_VEL
LIN {X 0,Y 146.659,Z 977.826,A -85,B 0,C 180,E1 7871.925,E2 7871.925} C_VEL
LIN {X 0,Y 138.287,Z 985.563,A -85,B 0,C 180,E1 7864.333,E2 7864.333} C_VEL
LIN {X 0,Y 132.175,Z 991.659,A -85,B 0,C 180,E1 7855.545,E2 7855.545} C_VEL
LIN {X 0,Y 129.048,Z 995.639,A -85,B 0,C 180,E1 7846.661,E2 7846.661} C_VEL
LIN {X 0,Y 128.273,Z 997.88,A -85,B 0,C 180,E1 7838.068,E2 7838.068} C_VEL
LIN {X 0,Y 128.485,Z 998.565,A -85,B 0,C 180,E1 7831.786,E2 7831.786} C_VEL
LIN {X 0,Y 128.407,Z 998.457,A -85,B 0,C 180,E1 7826.431,E2 7826.431} C_VEL
LIN {X 0,Y 128.328,Z 997.225,A -85,B 0,C 180,E1 7818.77,E2 7818.77} C_VEL
LIN {X 0,Y 129.958,Z 994.244,A -85,B 0,C 180,E1 7809.746,E2 7809.746} C_VEL
LIN {X 0,Y 134.394,Z 989.222,A -85,B 0,C 180,E1 7800.595,E2 7800.595} C_VEL
LIN {X 0,Y 141.302,Z 982.599,A -85,B 0,C 180,E1 7792.519,E2 7792.519} C_VEL
LIN {X 0,Y 150.094,Z 974.537,A -85,B 0,C 180,E1 7785.619,E2 7785.619} C_VEL
LIN {X 0,Y 160.766,Z 964.575,A -85,B 0,C 180,E1 7779.541,E2 7779.541} C_VEL
LIN {X 0,Y 172.341,Z 953.138,A -85,B 0,C 180,E1 7774.533,E2 7774.533} C_VEL
LIN {X 0,Y 184.346,Z 940.253,A -85,B 0,C 180,E1 7770.418,E2 7770.418} C_VEL
LIN {X 0,Y 196.437,Z 925.885,A -85,B 0,C 180,E1 7767.036,E2 7767.036} C_VEL
LIN {X 0,Y 208.355,Z 909.894,A -85,B 0,C 180,E1 7764.251,E2 7764.251} C_VEL
LIN {X 0,Y 219.415,Z 892.9,A -85,B 0,C 180,E1 7762.043,E2 7762.043} C_VEL
LIN {X 0,Y 229.238,Z 875.394,A -85,B 0,C 180,E1 7760.325,E2 7760.325} C_VEL
LIN {X 0,Y 237.9,Z 857.271,A -85,B 0,C 180,E1 7758.982,E2 7758.982} C_VEL
LIN {X 0,Y 245.834,Z 837.195,A -85,B 0,C 180,E1 7757.879,E2 7757.879} C_VEL
LIN {X 0,Y 252.089,Z 817.234,A -85,B 0,C 180,E1 7757.088,E2 7757.088} C_VEL
LIN {X 0,Y 256.853,Z 796.652,A -85,B 0,C 180,E1 7756.478,E2 7756.478} C_VEL
LIN {X 0,Y 259.934,Z 776.865,A -85,B 0,C 180,E1 7756.099,E2 7756.099} C_VEL
LIN {X 0,Y 262.187,Z 757.682,A -85,B 0,C 180,E1 7755.922,E2 7755.922} C_VEL
LIN {X 0,Y 261.761,Z 731.901,A -85,B 0,C 180,E1 7752.827,E2 7752.827} C_VEL
LIN {X 0,Y 262.434,Z 705,A -85,B 0,C 180,E1 7749.969,E2 7749.969} C_VEL
LIN {X 0,Y 263.761,Z 681.085,A -85,B 0,C 180,E1 7747.734,E2 7747.734} C_VEL
LIN {X 0,Y 263.269,Z 669.462,A -85,B 0,C 180,E1 7743.756,E2 7743.756} C_VEL
LIN {X 0,Y 264.344,Z 656.142,A -85,B 0,C 180,E1 7738.32,E2 7738.32} C_VEL
LIN {X 0,Y 266.5,Z 647.745,A -85,B 0,C 180,E1 7734.294,E2 7734.294} C_VEL
LIN {X 0,Y 267.831,Z 644.544,A -85,B 0,C 180,E1 7732.492,E2 7732.492} C_VEL
LIN {X 0,Y 268.898,Z 646.975,A -85,B 0,C 180,E1 7730.475,E2 7730.475} C_VEL
LIN {X 0,Y 271.051,Z 652.069,A -85,B 0,C 180,E1 7727.375,E2 7727.375} C_VEL
LIN {X 0,Y 272.514,Z 655.867,A -85,B 0,C 180,E1 7725.633,E2 7725.633} C_VEL
LIN {X 0,Y 259.721,Z 777.35,A -85,B 0,C 180,E1 7723.292,E2 7723.292} C_VEL
LIN {X 0,Y 256.04,Z 797.657,A -85,B 0,C 180,E1 7722.703,E2 7722.703} C_VEL
LIN {X 0,Y 250.839,Z 817.833,A -85,B 0,C 180,E1 7721.885,E2 7721.885} C_VEL
LIN {X 0,Y 244.055,Z 837.898,A -85,B 0,C 180,E1 7720.787,E2 7720.787} C_VEL
LIN {X 0,Y 236.454,Z 856.053,A -85,B 0,C 180,E1 7719.489,E2 7719.489} C_VEL
LIN {X 0,Y 227.714,Z 873.523,A -85,B 0,C 180,E1 7717.888,E2 7717.888} C_VEL
LIN {X 0,Y 217.115,Z 891.397,A -85,B 0,C 180,E1 7715.756,E2 7715.756} C_VEL
LIN {X 0,Y 206.043,Z 907.438,A -85,B 0,C 180,E1 7713.235,E2 7713.235} C_VEL
LIN {X 0,Y 194.628,Z 921.937,A -85,B 0,C 180,E1 7710.247,E2 7710.247} C_VEL
LIN {X 0,Y 183.068,Z 935.013,A -85,B 0,C 180,E1 7706.679,E2 7706.679} C_VEL
LIN {X 0,Y 170.799,Z 947.487,A -85,B 0,C 180,E1 7702.071,E2 7702.071} C_VEL
LIN {X 0,Y 159.436,Z 958.023,A -85,B 0,C 180,E1 7696.671,E2 7696.671} C_VEL
LIN {X 0,Y 149.439,Z 966.684,A -85,B 0,C 180,E1 7690.464,E2 7690.464} C_VEL
LIN {X 0,Y 140.799,Z 973.897,A -85,B 0,C 180,E1 7683.074,E2 7683.074} C_VEL
LIN {X 0,Y 134.258,Z 979.418,A -85,B 0,C 180,E1 7674.646,E2 7674.646} C_VEL
LIN {X 0,Y 130.247,Z 983.088,A -85,B 0,C 180,E1 7665.583,E2 7665.583} C_VEL
LIN {X 0,Y 128.645,Z 984.882,A -85,B 0,C 180,E1 7657.141,E2 7657.141} C_VEL
LIN {X 0,Y 128.358,Z 985.411,A -85,B 0,C 180,E1 7649.551,E2 7649.551} C_VEL
LIN {X 0,Y 128.732,Z 984.782,A -85,B 0,C 180,E1 7641.961,E2 7641.961} C_VEL
LIN {X 0,Y 130.64,Z 982.693,A -85,B 0,C 180,E1 7633.078,E2 7633.078} C_VEL
LIN {X 0,Y 134.729,Z 979.038,A -85,B 0,C 180,E1 7624.502,E2 7624.502} C_VEL
LIN {X 0,Y 141.557,Z 973.356,A -85,B 0,C 180,E1 7616.08,E2 7616.08} C_VEL
LIN {X 0,Y 150.706,Z 965.754,A -85,B 0,C 180,E1 7608.565,E2 7608.565} C_VEL
LIN {X 0,Y 161.085,Z 956.715,A -85,B 0,C 180,E1 7602.382,E2 7602.382} C_VEL
LIN {X 0,Y 172.172,Z 946.324,A -85,B 0,C 180,E1 7597.285,E2 7597.285} C_VEL
LIN {X 0,Y 183.681,Z 934.539,A -85,B 0,C 180,E1 7593.037,E2 7593.037} C_VEL
LIN {X 0,Y 188.021,Z 929.74,A -85,B 0,C 180,E1 7591.588,E2 7591.588} C_VEL
LIN {X 0,Y 172.993,Z 934.997,A -85,B 0,C 180,E1 7586.427,E2 7586.427} C_VEL
LIN {X 0,Y 162.383,Z 938.685,A -85,B 0,C 180,E1 7581.303,E2 7581.303} C_VEL
LIN {X 0,Y 153.798,Z 941.882,A -85,B 0,C 180,E1 7575.459,E2 7575.459} C_VEL
LIN {X 0,Y 147.125,Z 944.771,A -85,B 0,C 180,E1 7568.599,E2 7568.599} C_VEL
LIN {X 0,Y 142.988,Z 947.487,A -85,B 0,C 180,E1 7561.203,E2 7561.203} C_VEL
LIN {X 0,Y 141.614,Z 950.579,A -85,B 0,C 180,E1 7551.883,E2 7551.883} C_VEL
LIN {X 0,Y 145.73,Z 953.953,A -85,B 0,C 180,E1 7540.356,E2 7540.356} C_VEL
LIN {X 0,Y 156.426,Z 956.493,A -85,B 0,C 180,E1 7530.072,E2 7530.072} C_VEL
LIN {X 0,Y 157.934,Z 957.315,A -85,B 0,C 180,E1 7528.499,E2 7528.499} C_VEL
LIN {X 0,Y 158.319,Z 959.107,A -85,B 0,C 180,E1 7526.624,E2 7526.624} C_VEL
LIN {X 0,Y 157.16,Z 962.088,A -85,B 0,C 180,E1 7524.283,E2 7524.283} C_VEL
LIN {X 0,Y 154.773,Z 965.077,A -85,B 0,C 180,E1 7522.386,E2 7522.386} C_VEL
LIN {X 0,Y 153.966,Z 965.863,A -85,B 0,C 180,E1 7521.959,E2 7521.959} C_VEL
LIN {X 0,Y 143.27,Z 975.144,A -85,B 0,C 180,E1 7515.96,E2 7515.96} C_VEL
LIN {X 0,Y 133.598,Z 983.335,A -85,B 0,C 180,E1 7508.405,E2 7508.405} C_VEL
LIN {X 0,Y 126.129,Z 989.908,A -85,B 0,C 180,E1 7499.441,E2 7499.441} C_VEL
LIN {X 0,Y 121.73,Z 994.539,A -85,B 0,C 180,E1 7489.682,E2 7489.682} C_VEL
LIN {X 0,Y 120.308,Z 997.16,A -85,B 0,C 180,E1 7480.538,E2 7480.538} C_VEL
LIN {X 0,Y 120.45,Z 998.102,A -85,B 0,C 180,E1 7472.857,E2 7472.857} C_VEL
LIN {X 0,Y 120.467,Z 998.123,A -85,B 0,C 180,E1 7467.624,E2 7467.624} C_VEL
LIN {X 0,Y 120.265,Z 997.298,A -85,B 0,C 180,E1 7460.431,E2 7460.431} C_VEL
LIN {X 0,Y 121.576,Z 994.677,A -85,B 0,C 180,E1 7450.797,E2 7450.797} C_VEL
LIN {X 0,Y 125.896,Z 990.052,A -85,B 0,C 180,E1 7440.88,E2 7440.88} C_VEL
LIN {X 0,Y 133.132,Z 983.634,A -85,B 0,C 180,E1 7431.99,E2 7431.99} C_VEL
LIN {X 0,Y 142.309,Z 975.858,A -85,B 0,C 180,E1 7424.635,E2 7424.635} C_VEL
LIN {X 0,Y 153.528,Z 966.113,A -85,B 0,C 180,E1 7418.22,E2 7418.22} C_VEL
LIN {X 0,Y 165.709,Z 954.823,A -85,B 0,C 180,E1 7413,E2 7413} C_VEL
LIN {X 0,Y 178.061,Z 942.266,A -85,B 0,C 180,E1 7408.843,E2 7408.843} C_VEL
LIN {X 0,Y 190.025,Z 928.795,A -85,B 0,C 180,E1 7405.56,E2 7405.56} C_VEL
LIN {X 0,Y 202.076,Z 913.598,A -85,B 0,C 180,E1 7402.807,E2 7402.807} C_VEL
LIN {X 0,Y 213.581,Z 897.051,A -85,B 0,C 180,E1 7400.568,E2 7400.568} C_VEL
LIN {X 0,Y 223.932,Z 879.852,A -85,B 0,C 180,E1 7398.816,E2 7398.816} C_VEL
LIN {X 0,Y 233.177,Z 861.854,A -85,B 0,C 180,E1 7397.436,E2 7397.436} C_VEL
LIN {X 0,Y 241.679,Z 841.809,A -85,B 0,C 180,E1 7396.303,E2 7396.303} C_VEL
LIN {X 0,Y 248.341,Z 822.1,A -85,B 0,C 180,E1 7395.498,E2 7395.498} C_VEL
LIN {X 0,Y 253.56,Z 801.707,A -85,B 0,C 180,E1 7394.886,E2 7394.886} C_VEL
LIN {X 0,Y 257.189,Z 781.054,A -85,B 0,C 180,E1 7394.446,E2 7394.446} C_VEL
LIN {X 0,Y 259.823,Z 759.73,A -85,B 0,C 180,E1 7394.24,E2 7394.24} C_VEL
LIN {X 0,Y 259.861,Z 732.387,A -85,B 0,C 180,E1 7390.951,E2 7390.951} C_VEL
LIN {X 0,Y 261.054,Z 704.738,A -85,B 0,C 180,E1 7388.077,E2 7388.077} C_VEL
LIN {X 0,Y 262.298,Z 686.306,A -85,B 0,C 180,E1 7386.346,E2 7386.346} C_VEL
LIN {X 0,Y 262.179,Z 676.206,A -85,B 0,C 180,E1 7382.841,E2 7382.841} C_VEL
LIN {X 0,Y 263.578,Z 663.288,A -85,B 0,C 180,E1 7377.554,E2 7377.554} C_VEL
LIN {X 0,Y 265.903,Z 655.106,A -85,B 0,C 180,E1 7373.631,E2 7373.631} C_VEL
LIN {X 0,Y 266.899,Z 652.718,A -85,B 0,C 180,E1 7372.357,E2 7372.357} C_VEL
LIN {X 0,Y 268.615,Z 657.102,A -85,B 0,C 180,E1 7369.274,E2 7369.274} C_VEL
LIN {X 0,Y 270.111,Z 661.113,A -85,B 0,C 180,E1 7367.185,E2 7367.185} C_VEL
LIN {X 0,Y 257.509,Z 777.881,A -85,B 0,C 180,E1 7364.992,E2 7364.992} C_VEL
LIN {X 0,Y 253.75,Z 798.149,A -85,B 0,C 180,E1 7364.423,E2 7364.423} C_VEL
LIN {X 0,Y 248.458,Z 818.248,A -85,B 0,C 180,E1 7363.638,E2 7363.638} C_VEL
LIN {X 0,Y 241.538,Z 838.291,A -85,B 0,C 180,E1 7362.582,E2 7362.582} C_VEL
LIN {X 0,Y 233.764,Z 856.453,A -85,B 0,C 180,E1 7361.33,E2 7361.33} C_VEL
LIN {X 0,Y 224.813,Z 873.927,A -85,B 0,C 180,E1 7359.785,E2 7359.785} C_VEL
LIN {X 0,Y 214.293,Z 891.238,A -85,B 0,C 180,E1 7357.794,E2 7357.794} C_VEL
LIN {X 0,Y 203.34,Z 906.761,A -85,B 0,C 180,E1 7355.457,E2 7355.457} C_VEL
LIN {X 0,Y 191.518,Z 921.443,A -85,B 0,C 180,E1 7352.56,E2 7352.56} C_VEL
LIN {X 0,Y 179.476,Z 934.675,A -85,B 0,C 180,E1 7349.082,E2 7349.082} C_VEL
LIN {X 0,Y 167.466,Z 946.508,A -85,B 0,C 180,E1 7344.878,E2 7344.878} C_VEL
LIN {X 0,Y 155.804,Z 956.942,A -85,B 0,C 180,E1 7339.786,E2 7339.786} C_VEL
LIN {X 0,Y 144.397,Z 966.319,A -85,B 0,C 180,E1 7333.273,E2 7333.273} C_VEL
LIN {X 0,Y 134.54,Z 973.977,A -85,B 0,C 180,E1 7325.425,E2 7325.425} C_VEL
LIN {X 0,Y 127.222,Z 979.604,A -85,B 0,C 180,E1 7316.611,E2 7316.611} C_VEL
LIN {X 0,Y 122.802,Z 983.201,A -85,B 0,C 180,E1 7307.53,E2 7307.53} C_VEL
LIN {X 0,Y 120.748,Z 985.232,A -85,B 0,C 180,E1 7298.09,E2 7298.09} C_VEL
LIN {X 0,Y 120.374,Z 985.833,A -85,B 0,C 180,E1 7289.997,E2 7289.997} C_VEL
LIN {X 0,Y 120.74,Z 985.258,A -85,B 0,C 180,E1 7281.905,E2 7281.905} C_VEL
LIN {X 0,Y 122.625,Z 983.414,A -85,B 0,C 180,E1 7272.928,E2 7272.928} C_VEL
LIN {X 0,Y 127.179,Z 979.698,A -85,B 0,C 180,E1 7263.374,E2 7263.374} C_VEL
LIN {X 0,Y 134.481,Z 974.089,A -85,B 0,C 180,E1 7254.552,E2 7254.552} C_VEL
LIN {X 0,Y 143.801,Z 966.857,A -85,B 0,C 180,E1 7247.044,E2 7247.044} C_VEL
LIN {X 0,Y 154.504,Z 958.128,A -85,B 0,C 180,E1 7240.783,E2 7240.783} C_VEL
LIN {X 0,Y 166.027,Z 947.975,A -85,B 0,C 180,E1 7235.606,E2 7235.606} C_VEL
LIN {X 0,Y 177.921,Z 936.455,A -85,B 0,C 180,E1 7231.326,E2 7231.326} C_VEL
LIN {X 0,Y 167.744,Z 939.812,A -85,B 0,C 180,E1 7227.706,E2 7227.706} C_VEL
LIN {X 0,Y 157.262,Z 943.153,A -85,B 0,C 180,E1 7222.82,E2 7222.82} C_VEL
LIN {X 0,Y 147.784,Z 946.388,A -85,B 0,C 180,E1 7216.509,E2 7216.509} C_VEL
LIN {X 0,Y 141.005,Z 949.155,A -85,B 0,C 180,E1 7209.709,E2 7209.709} C_VEL
LIN {X 0,Y 136.381,Z 951.844,A -85,B 0,C 180,E1 7201.681,E2 7201.681} C_VEL
LIN {X 0,Y 134.824,Z 954.81,A -85,B 0,C 180,E1 7191.901,E2 7191.901} C_VEL
LIN {X 0,Y 139.059,Z 958.159,A -85,B 0,C 180,E1 7179.811,E2 7179.811} C_VEL
LIN {X 0,Y 154.102,Z 961.198,A -85,B 0,C 180,E1 7166.53,E2 7166.53} C_VEL
LIN {X 0,Y 158.57,Z 961.664,A -85,B 0,C 180,E1 7164.098,E2 7164.098} C_VEL
LIN {X 0,Y 153.966,Z 965.863,A -85,B 0,C 180,E1 7161.959,E2 7161.959} C_VEL
LIN {X 0,Y 149.143,Z 969.55,A -85,B 0,C 180,E1 7160.129,E2 7160.129} C_VEL
LIN {X 0,Y 134.546,Z 977.812,A -85,B 0,C 180,E1 7155.613,E2 7155.613} C_VEL
LIN {X 0,Y 130.11,Z 980.717,A -85,B 0,C 180,E1 7153.158,E2 7153.158} C_VEL
LIN {X 0,Y 121.06,Z 987.865,A -85,B 0,C 180,E1 7144.171,E2 7144.171} C_VEL
LIN {X 0,Y 115.153,Z 993.018,A -85,B 0,C 180,E1 7134.088,E2 7134.088} C_VEL
LIN {X 0,Y 112.568,Z 996.167,A -85,B 0,C 180,E1 7123.879,E2 7123.879} C_VEL
LIN {X 0,Y 112.377,Z 997.607,A -85,B 0,C 180,E1 7114.596,E2 7114.596} C_VEL
LIN {X 0,Y 112.509,Z 997.762,A -85,B 0,C 180,E1 7108.475,E2 7108.475} C_VEL
LIN {X 0,Y 112.265,Z 997.109,A -85,B 0,C 180,E1 7101.294,E2 7101.294} C_VEL
LIN {X 0,Y 113.343,Z 994.935,A -85,B 0,C 180,E1 7091.486,E2 7091.486} C_VEL
LIN {X 0,Y 117.279,Z 990.986,A -85,B 0,C 180,E1 7081.415,E2 7081.415} C_VEL
LIN {X 0,Y 124.551,Z 984.975,A -85,B 0,C 180,E1 7071.823,E2 7071.823} C_VEL
LIN {X 0,Y 134.252,Z 977.317,A -85,B 0,C 180,E1 7063.749,E2 7063.749} C_VEL
LIN {X 0,Y 145.548,Z 968.172,A -85,B 0,C 180,E1 7057.171,E2 7057.171} C_VEL
LIN {X 0,Y 157.764,Z 957.628,A -85,B 0,C 180,E1 7051.874,E2 7051.874} C_VEL
LIN {X 0,Y 170.378,Z 945.743,A -85,B 0,C 180,E1 7047.612,E2 7047.612} C_VEL
LIN {X 0,Y 183.008,Z 932.539,A -85,B 0,C 180,E1 7044.165,E2 7044.165} C_VEL
LIN {X 0,Y 195.837,Z 917.402,A -85,B 0,C 180,E1 7041.293,E2 7041.293} C_VEL
LIN {X 0,Y 207.818,Z 901.182,A -85,B 0,C 180,E1 7039.025,E2 7039.025} C_VEL
LIN {X 0,Y 218.122,Z 885.115,A -85,B 0,C 180,E1 7037.334,E2 7037.334} C_VEL
LIN {X 0,Y 228.176,Z 866.848,A -85,B 0,C 180,E1 7035.884,E2 7035.884} C_VEL
LIN {X 0,Y 236.799,Z 848.144,A -85,B 0,C 180,E1 7034.782,E2 7034.782} C_VEL
LIN {X 0,Y 243.894,Z 829.386,A -85,B 0,C 180,E1 7033.964,E2 7033.964} C_VEL
LIN {X 0,Y 250.057,Z 808.27,A -85,B 0,C 180,E1 7033.297,E2 7033.297} C_VEL
LIN {X 0,Y 254.46,Z 786.611,A -85,B 0,C 180,E1 7032.789,E2 7032.789} C_VEL
LIN {X 0,Y 257.691,Z 761.689,A -85,B 0,C 180,E1 7032.521,E2 7032.521} C_VEL
LIN {X 0,Y 258.202,Z 734.138,A -85,B 0,C 180,E1 7029.205,E2 7029.205} C_VEL
LIN {X 0,Y 259.865,Z 705.661,A -85,B 0,C 180,E1 7026.267,E2 7026.267} C_VEL
LIN {X 0,Y 260.991,Z 691.529,A -85,B 0,C 180,E1 7024.945,E2 7024.945} C_VEL
LIN {X 0,Y 261.164,Z 682.813,A -85,B 0,C 180,E1 7021.864,E2 7021.864} C_VEL
LIN {X 0,Y 262.859,Z 670.433,A -85,B 0,C 180,E1 7016.783,E2 7016.783} C_VEL
LIN {X 0,Y 265.424,Z 662.276,A -85,B 0,C 180,E1 7012.859,E2 7012.859} C_VEL
LIN {X 0,Y 265.999,Z 661.18,A -85,B 0,C 180,E1 7012.114,E2 7012.114} C_VEL
LIN {X 0,Y 267.813,Z 666.05,A -85,B 0,C 180,E1 7008.914,E2 7008.914} C_VEL
LIN {X 0,Y 267.877,Z 666.668,A -85,B 0,C 180,E1 7008.757,E2 7008.757} C_VEL
LIN {X 0,Y 255.542,Z 778.313,A -85,B 0,C 180,E1 7006.721,E2 7006.721} C_VEL
LIN {X 0,Y 251.692,Z 798.641,A -85,B 0,C 180,E1 7006.173,E2 7006.173} C_VEL
LIN {X 0,Y 246.314,Z 818.66,A -85,B 0,C 180,E1 7005.423,E2 7005.423} C_VEL
LIN {X 0,Y 239.262,Z 838.683,A -85,B 0,C 180,E1 7004.413,E2 7004.413} C_VEL
LIN {X 0,Y 231.321,Z 856.852,A -85,B 0,C 180,E1 7003.213,E2 7003.213} C_VEL
LIN {X 0,Y 222.164,Z 874.33,A -85,B 0,C 180,E1 7001.73,E2 7001.73} C_VEL
LIN {X 0,Y 211.227,Z 891.886,A -85,B 0,C 180,E1 6999.784,E2 6999.784} C_VEL
LIN {X 0,Y 199.713,Z 907.715,A -85,B 0,C 180,E1 6997.469,E2 6997.469} C_VEL
LIN {X 0,Y 187.932,Z 921.856,A -85,B 0,C 180,E1 6994.746,E2 6994.746} C_VEL
LIN {X 0,Y 175.454,Z 935.09,A -85,B 0,C 180,E1 6991.35,E2 6991.35} C_VEL
LIN {X 0,Y 162.937,Z 946.925,A -85,B 0,C 180,E1 6987.211,E2 6987.211} C_VEL
LIN {X 0,Y 150.69,Z 957.359,A -85,B 0,C 180,E1 6982.144,E2 6982.144} C_VEL
LIN {X 0,Y 138.594,Z 966.737,A -85,B 0,C 180,E1 6975.576,E2 6975.576} C_VEL
LIN {X 0,Y 128.011,Z 974.396,A -85,B 0,C 180,E1 6967.531,E2 6967.531} C_VEL
LIN {X 0,Y 120.033,Z 980.021,A -85,B 0,C 180,E1 6958.344,E2 6958.344} C_VEL
LIN {X 0,Y 115.133,Z 983.617,A -85,B 0,C 180,E1 6948.74,E2 6948.74} C_VEL
LIN {X 0,Y 112.815,Z 985.645,A -85,B 0,C 180,E1 6938.663,E2 6938.663} C_VEL
LIN {X 0,Y 112.384,Z 986.244,A -85,B 0,C 180,E1 6929.997,E2 6929.997} C_VEL
LIN {X 0,Y 112.807,Z 985.671,A -85,B 0,C 180,E1 6921.331,E2 6921.331} C_VEL
LIN {X 0,Y 114.936,Z 983.829,A -85,B 0,C 180,E1 6911.747,E2 6911.747} C_VEL
LIN {X 0,Y 119.99,Z 980.114,A -85,B 0,C 180,E1 6901.639,E2 6901.639} C_VEL
LIN {X 0,Y 127.952,Z 974.506,A -85,B 0,C 180,E1 6892.442,E2 6892.442} C_VEL
LIN {X 0,Y 138.296,Z 967.041,A -85,B 0,C 180,E1 6884.532,E2 6884.532} C_VEL
LIN {X 0,Y 149.326,Z 958.543,A -85,B 0,C 180,E1 6878.423,E2 6878.423} C_VEL
LIN {X 0,Y 161.441,Z 948.388,A -85,B 0,C 180,E1 6873.266,E2 6873.266} C_VEL
LIN {X 0,Y 167.409,Z 942.916,A -85,B 0,C 180,E1 6871.033,E2 6871.033} C_VEL
LIN {X 0,Y 152.16,Z 947.463,A -85,B 0,C 180,E1 6864.456,E2 6864.456} C_VEL
LIN {X 0,Y 142.115,Z 950.561,A -85,B 0,C 180,E1 6858.034,E2 6858.034} C_VEL
LIN {X 0,Y 134.614,Z 953.334,A -85,B 0,C 180,E1 6850.702,E2 6850.702} C_VEL
LIN {X 0,Y 129.805,Z 955.925,A -85,B 0,C 180,E1 6842.65,E2 6842.65} C_VEL
LIN {X 0,Y 127.928,Z 958.865,A -85,B 0,C 180,E1 6831.913,E2 6831.913} C_VEL
LIN {X 0,Y 132.243,Z 962.079,A -85,B 0,C 180,E1 6819.186,E2 6819.186} C_VEL
LIN {X 0,Y 147.796,Z 965.106,A -85,B 0,C 180,E1 6805.371,E2 6805.371} C_VEL
LIN {X 0,Y 149.183,Z 965.31,A -85,B 0,C 180,E1 6804.524,E2 6804.524} C_VEL
LIN {X 0,Y 137.666,Z 974.722,A -85,B 0,C 180,E1 6798.428,E2 6798.428} C_VEL
LIN {X 0,Y 130.11,Z 980.717,A -85,B 0,C 180,E1 6793.158,E2 6793.158} C_VEL
LIN {X 0,Y 125.883,Z 983.439,A -85,B 0,C 180,E1 6790.505,E2 6790.505} C_VEL
LIN {X 0,Y 113.11,Z 989.112,A -85,B 0,C 180,E1 6783.529,E2 6783.529} C_VEL
LIN {X 0,Y 109.807,Z 990.867,A -85,B 0,C 180,E1 6780.021,E2 6780.021} C_VEL
LIN {X 0,Y 105.382,Z 994.88,A -85,B 0,C 180,E1 6768.823,E2 6768.823} C_VEL
LIN {X 0,Y 104.291,Z 996.858,A -85,B 0,C 180,E1 6758.271,E2 6758.271} C_VEL
LIN {X 0,Y 104.548,Z 997.403,A -85,B 0,C 180,E1 6750.551,E2 6750.551} C_VEL
LIN {X 0,Y 104.293,Z 997.068,A -85,B 0,C 180,E1 6743.397,E2 6743.397} C_VEL
LIN {X 0,Y 104.912,Z 995.353,A -85,B 0,C 180,E1 6733.39,E2 6733.39} C_VEL
